(* IEC 61131-3 sources: Codesys/60-let-oktyabrya/src (part 2) *)

(* ---- PRG_AlarmLogSD.st ---- *)
(* ============================================================ *)
(* PRG_AlarmLogSD — ЖУРНАЛЫ НА SD-КАРТУ (3 файла В МЕСЯЦ)        *)
(* ============================================================ *)
(* Пишет на SD три отдельных журнала (чтобы записи не путались): *)
(*   • АВАРИИ     → sAlarmLogPath   (alarms-MM-YYYY.log)         *)
(*   • ИЗМЕНЕНИЯ ПЧ→ sPumpLogPath    (pump_changes-MM-YYYY.log)  *)
(*   • УСТАВКИ    → sSetpointLogPath (setpoints-MM-YYYY.log)     *)
(*                                                              *)
(* === НОВОЕ: ПОМЕСЯЧНЫЕ ФАЙЛЫ ==============================    *)
(* Имя файла содержит месяц и год, поэтому 1-го числа нового     *)
(* месяца путь меняется САМ, и старый автомат (OPEN → если нет   *)
(* файла, то CREATE + BOM) создаёт новый файл без единой строчки *)
(* дополнительной логики. Отдельного «переключателя месяца» нет  *)
(* специально: любая пропущенная граница (ПЛК был выключен,      *)
(* карту вынимали) отрабатывается сама собой при первой записи.  *)
(*                                                              *)
(* === НОВОЕ: КОНТРОЛЬ МЕСТА ================================    *)
(* FB_SdSpaceGuard раз в tSdCheckPeriod (по умолчанию час), при  *)
(* смене месяца и после серии неудачных записей удаляет три файла *)
(* самого старого месяца, если журналы переросли квоту:            *)
(*     квота = ёмкость карты − 100 МБ резерва − чужие файлы        *)
(* Файл текущего месяца удалить нельзя ни при каких условиях.      *)
(*                                                               *)
(* ЁМКОСТЬ КАРТЫ ОПРЕДЕЛЯЕТСЯ АВТОМАТИЧЕСКИ — FB_SdCardSize        *)
(* читает размер раздела у ядра (/sys/block/...). Номинал из       *)
(* выпадающего списка на экране (iSdCardSize) — только запасной    *)
(* вариант, если автоопределение не сработало. Кнопок нет.         *)
(*                                                              *)
(* Строка: "чч:мм дд.мм.гггг - текст" (для аварий) либо готовая  *)
(* строка журнала (для ПЧ/уставок). WSTRING/UTF-16LE + BOM.     *)
(*                                                              *)
(* Аварии детектируются здесь СТРОГО ПО ФРОНТУ FALSE→TRUE: пока  *)
(* авария висит, повторных записей нет. Изменения ПЧ/уставок     *)
(* кладут строку в глобальные очереди GVL_Fountain.awsSdPumpQ /  *)
(* awsSdSetpQ прямо из F_PumpLogWrite / F_FountainLogWrite —      *)
(* здесь мы их только забираем и пишем в файл.                   *)
(*                                                              *)
(* Один конечный автомат обслуживает по очереди все три файла    *)
(* (приоритет: аварии → ПЧ → уставки). ФБ CAA File асинхронные.  *)
(* Пока сторож места занят (fbGuard.xBusy) — новая строка не     *)
(* начинается, строки ждут в очередях.                           *)
(*                                                              *)
(* ТРЕБОВАНИЯ: библиотека CAA File (тип FILE.CAA.HANDLE), карта   *)
(* SD FAT16/FAT32 MBR, путь /mnt/ufs/media/mmcblk0p1/.           *)
(* ============================================================ *)
PROGRAM PRG_AlarmLogSD
VAR CONSTANT
    cAlarmCnt       : INT := 11;   // сколько аварий отслеживаем
    cQSize          : INT := 20;   // глубина очереди строк
    cWriteFailForce : INT := 3;    // столько неудачных записей подряд =
                                   // карта полна → удалить старый месяц
END_VAR
VAR
    (* --- Аварии: состояние + названия --- *)
    axAlarmNow  : ARRAY[1..cAlarmCnt] OF BOOL;
    axAlarmPrev : ARRAY[1..cAlarmCnt] OF BOOL;
    awsAlarmName : ARRAY[1..cAlarmCnt] OF WSTRING(60) := [
        "Сухой ход",
        "Сухой ход реле",
        "Клапан добора реле",
        "Насосы фонтана реле",
        "Подсветка реле",
        "Фильтрация реле (ручной режим)",
        "Связь ПЧ1",
        "Связь ПЧ2",
        "Связь ПЧ3",
        "Связь МВ-Д",
        "Связь МУ"];

    (* --- Локальная очередь аварий (сырые строки, без CRLF) --- *)
    awsAlarmQ : ARRAY[1..cQSize] OF WSTRING(120);
    iAQHead : INT;  iAQTail : INT;  iAQCount : INT;

    (* --- Конечный автомат записи --- *)
    iState     : INT;   // 0=IDLE 1=OPEN 2=CREATE 6=BOM 3=WRITE 4=FLUSH 5=CLOSE 9=DROP
    wsLineOut  : WSTRING(122);
    sActivePath : STRING(80);
    wBom       : WORD := 16#FEFF;   // BOM UTF-16LE (байты FF FE)

    (* --- ФБ CAA File --- *)
    fbFileOpen  : FILE.Open;
    fbFileWrite : FILE.Write;
    fbFileFlush : FILE.Flush;
    fbFileClose : FILE.Close;
    hFile       : FILE.CAA.HANDLE;

    iWrittenCnt : INT;
    iDroppedCnt : INT;

    i          : INT;
    wsTimeStamp : WSTRING(24);
    wsHH : WSTRING(4);  wsMM : WSTRING(4);
    wsDD : WSTRING(4);  wsMo : WSTRING(4);  wsYY : WSTRING(6);

    (* --- Помесячные файлы --- *)
    iLogYear      : INT;    // год/месяц, в которые сейчас пишем
    iLogMonth     : INT;
    iLogYearPrev  : INT;    // 0 при старте → пути соберутся в 1-м же цикле
    iLogMonthPrev : INT;

    (* --- Сторож места на карте --- *)
    fbGuard         : FB_SdSpaceGuard;
    fbCardSize      : FB_SdCardSize;   // автоопределение ёмкости карты
    tonSdCheck      : TON;
    xGuardTrig      : BOOL;
    xGuardStart     : BOOL;
    xCapTrig        : BOOL;   // перечитать ёмкость карты
    xGuardForceAuto : BOOL;   // авто-форс: карта полна (серия отказов записи)
    iWriteFailCnt   : INT;    // неудачных записей подряд
END_VAR

(* ============================================================ *)
(* 1. КАРТА АВАРИЙ (порядок = порядок названий)                 *)
(* ============================================================ *)
axAlarmNow[1]  := xDryRunAlarm;
axAlarmNow[2]  := xDryRunRelayAlarm;
axAlarmNow[3]  := xDamperRelayAlarm;
axAlarmNow[4]  := xPumpRelayAlarm;
axAlarmNow[5]  := xLightRelayAlarm;
axAlarmNow[6]  := xNfManualRelayAlarm;
axAlarmNow[7]  := xPumpCommError[1];
axAlarmNow[8]  := xPumpCommError[2];
axAlarmNow[9]  := xPumpCommError[3];
axAlarmNow[10] := xMV110_Error;
axAlarmNow[11] := xMU110_Error;

(* ============================================================ *)
(* 2. МЕТКА ВРЕМЕНИ "чч:мм дд.мм.гггг"                          *)
(* ============================================================ *)
wsHH := INT_TO_WSTRING(iCurrentHour);   IF iCurrentHour   < 10 THEN wsHH := WCONCAT("0", wsHH); END_IF;
wsMM := INT_TO_WSTRING(iCurrentMinute); IF iCurrentMinute < 10 THEN wsMM := WCONCAT("0", wsMM); END_IF;
wsDD := INT_TO_WSTRING(iCurrentDay);    IF iCurrentDay    < 10 THEN wsDD := WCONCAT("0", wsDD); END_IF;
wsMo := INT_TO_WSTRING(iCurrentMonth);  IF iCurrentMonth  < 10 THEN wsMo := WCONCAT("0", wsMo); END_IF;
wsYY := INT_TO_WSTRING(iCurrentYear);
wsTimeStamp := WCONCAT(wsHH, WCONCAT(":", WCONCAT(wsMM, WCONCAT(" ",
               WCONCAT(wsDD, WCONCAT(".", WCONCAT(wsMo, WCONCAT(".", wsYY))))))));

(* ============================================================ *)
(* 3. ФРОНТ АВАРИИ → строка в локальную очередь аварий          *)
(* ============================================================ *)
FOR i := 1 TO cAlarmCnt DO
    IF axAlarmNow[i] AND NOT axAlarmPrev[i] THEN
        IF xAlarmLogSDEnable THEN
            IF iAQCount < cQSize THEN
                iAQTail := (iAQTail MOD cQSize) + 1;
                awsAlarmQ[iAQTail] := WCONCAT(wsTimeStamp, WCONCAT(" - ", awsAlarmName[i]));
                iAQCount := iAQCount + 1;
            ELSE
                iDroppedCnt := iDroppedCnt + 1;
            END_IF;
        END_IF;
    END_IF;
    axAlarmPrev[i] := axAlarmNow[i];
END_FOR;

(* ============================================================ *)
(* 4. ПУТИ ФАЙЛОВ ТЕКУЩЕГО МЕСЯЦА                               *)
(* ============================================================ *)
(* Если RTC ещё не готов или сбит (села батарейка) — год выйдет  *)
(* за 2000..2199. Писать в "alarms-01-1970.log" нельзя (такой     *)
(* месяц не разберётся обратно и файл станет неудаляемым), поэтому*)
(* весь «бесчасовой» период сваливаем в один файл 01-2000. Он     *)
(* заведомо самый старый по ключу, то есть удалится первым, когда *)
(* место кончится, — и при этом защищён как «текущий», пока RTC   *)
(* не починят.                                                   *)
IF iCurrentYear >= 2000 AND iCurrentYear <= 2199
   AND iCurrentMonth >= 1 AND iCurrentMonth <= 12 THEN
    iLogYear  := iCurrentYear;
    iLogMonth := iCurrentMonth;
    xSdRtcBad := FALSE;
ELSE
    iLogYear  := 2000;
    iLogMonth := 1;
    xSdRtcBad := TRUE;
END_IF;

IF iLogYear <> iLogYearPrev OR iLogMonth <> iLogMonthPrev THEN
    sAlarmLogPath    := F_SdLogPath(sSdLogDir, sAlarmLogPrefix, iLogYear, iLogMonth);
    sPumpLogPath     := F_SdLogPath(sSdLogDir, sPumpLogPrefix,  iLogYear, iLogMonth);
    sSetpointLogPath := F_SdLogPath(sSdLogDir, sSetpLogPrefix,  iLogYear, iLogMonth);
    iLogYearPrev     := iLogYear;
    iLogMonthPrev    := iLogMonth;
    xGuardTrig       := TRUE;    // новый месяц — сразу проверить место
    xCapTrig         := TRUE;    // и заодно перечитать ёмкость карты
END_IF;

(* ============================================================ *)
(* 5. СТОРОЖ МЕСТА НА КАРТЕ                                     *)
(* ============================================================ *)
(* Периодический тик (самосброс: Q взводится на 1 цикл за период) *)
tonSdCheck(IN := NOT tonSdCheck.Q, PT := tSdCheckPeriod);
IF tonSdCheck.Q THEN
    xCapTrig   := TRUE;
    xGuardTrig := TRUE;
END_IF;

(* --- ЁМКОСТЬ КАРТЫ ---                                           *)
(* Сначала пробуем определить её САМИ (FB_SdCardSize читает размер *)
(* раздела у ядра). Получилось — номинал из списка не нужен вообще. *)
(* Не получилось — берём выбранный на экране номинал.               *)
fbCardSize(xTrigger := xCapTrig AND (iState = 0) AND NOT fbGuard.xBusy,
           sSysPath := sSdCardSysPath);
IF fbCardSize.xBusy THEN
    xCapTrig := FALSE;
END_IF;

xSdCapAuto       := fbCardSize.xValid;
udiSdCapAutoMB   := fbCardSize.udiCapacityMB;
udiSdCardSectors := fbCardSize.udiSectors;

IF iSdCardSize < 0 THEN iSdCardSize := 0; END_IF;
IF iSdCardSize > 6 THEN iSdCardSize := 6; END_IF;

IF xSdCapAuto THEN
    udiSdUsableMB := udiSdCapAutoMB;
ELSE
    udiSdUsableMB := audiSdCardMB[iSdCardSize];
END_IF;

(* АВАРИЙНЫЙ ФОРС. Если запись не проходит подряд cWriteFailForce  *)
(* раз — карта реально полна, что бы ни говорил расчёт по номиналу *)
(* (например, в списке выбрали 32 ГБ, а стоит карта на 16). Тогда  *)
(* удаляем самый старый месяц безусловно. Одиночный сбой записи к  *)
(* удалению НЕ приводит — только серия подряд.                     *)
IF iWriteFailCnt >= cWriteFailForce THEN
    xGuardTrig      := TRUE;
    xGuardForceAuto := TRUE;
    iWriteFailCnt   := 0;
END_IF;

(* Запускаем сторожа ТОЛЬКО когда автомат записи стоит в IDLE:     *)
(* так исключено удаление файла при открытом дескрипторе.          *)
xGuardStart := xGuardTrig AND xAlarmLogSDEnable
               AND (iState = 0) AND NOT fbGuard.xBusy AND NOT fbCardSize.xBusy;

fbGuard(xTrigger      := xGuardStart,
        xForce        := xGuardForceAuto,
        sDir          := sSdLogDir,
        sPrefix1      := sAlarmLogPrefix,
        sPrefix2      := sPumpLogPrefix,
        sPrefix3      := sSetpLogPrefix,
        udiUsableMB   := udiSdUsableMB,
        udiFreeMinMB  := udiSdFreeMinMB,
        iCurYear      := iLogYear,
        iCurMonth     := iLogMonth);

IF fbGuard.xBusy THEN
    xGuardTrig      := FALSE;
    xGuardForceAuto := FALSE;
END_IF;

(* Диагностика на экран *)
udiSdQuotaMB       := fbGuard.udiQuotaMB;
udiSdOursMB        := fbGuard.udiOursMB;
udiSdUsedMB        := fbGuard.udiUsedMB;
udiSdForeignMB     := fbGuard.udiForeignMB;
udiSdOldestMB      := fbGuard.udiOldestMB;
xSdNothingToDelete := fbGuard.xNothingToDelete;
xSdLogQuotaStop    := fbGuard.xQuotaStop;
xSdCleanupFault    := fbGuard.xFault;
iSdDeletedTotal    := fbGuard.iDeletedTotal;
sSdLastDeleted     := fbGuard.sLastDeleted;

(* ============================================================ *)
(* 6. КОНЕЧНЫЙ АВТОМАТ: пишет по очереди 3 файла                *)
(*    приоритет: аварии → изменения ПЧ → уставки               *)
(* ============================================================ *)
(* Запись стоит, пока сторож занят (иначе он удалял бы файл с    *)
(* открытым дескриптором) ИЛИ пока поднят xQuotaStop — последний *)
(* рубеж защиты карты: наши журналы упёрлись в квоту, а удалять   *)
(* уже нечего. Строки при этом копятся в очередях, лишние         *)
(* считаются в iDroppedCnt; журналы на экране ведутся как обычно. *)
IF NOT fbGuard.xBusy AND NOT fbCardSize.xBusy AND NOT fbGuard.xQuotaStop THEN

CASE iState OF

    0:  (* IDLE — выбрать непустую очередь, взять строку, начать *)
        IF xAlarmLogSDEnable THEN
            IF iAQCount > 0 THEN
                iAQHead := (iAQHead MOD cQSize) + 1;
                wsLineOut := WCONCAT(awsAlarmQ[iAQHead], "$R$N");
                iAQCount := iAQCount - 1;
                sActivePath := sAlarmLogPath;
                iState := 1;
            ELSIF iSdPumpQCount > 0 THEN
                iSdPumpQHead := (iSdPumpQHead MOD 20) + 1;
                wsLineOut := WCONCAT(awsSdPumpQ[iSdPumpQHead], "$R$N");
                iSdPumpQCount := iSdPumpQCount - 1;
                sActivePath := sPumpLogPath;
                iState := 1;
            ELSIF iSdSetpQCount > 0 THEN
                iSdSetpQHead := (iSdSetpQHead MOD 20) + 1;
                wsLineOut := WCONCAT(awsSdSetpQ[iSdSetpQHead], "$R$N");
                iSdSetpQCount := iSdSetpQCount - 1;
                sActivePath := sSetpointLogPath;
                iState := 1;
            END_IF;
        END_IF;

    1:  (* OPEN на дозапись *)
        fbFileOpen(xExecute := TRUE, sFileName := sActivePath, eFileMode := FILE.MODE.MAPPD);
        IF fbFileOpen.xDone THEN
            hFile := fbFileOpen.hFile;
            fbFileOpen(xExecute := FALSE);
            iState := 3;
        ELSIF fbFileOpen.xError THEN
            IF fbFileOpen.eError = FILE.ERROR.NOT_EXIST THEN
                fbFileOpen(xExecute := FALSE);
                iState := 2;
            ELSE
                fbFileOpen(xExecute := FALSE);
                iState := 9;
            END_IF;
        END_IF;

    2:  (* CREATE — MWRITE создаёт файл *)
        fbFileOpen(xExecute := TRUE, sFileName := sActivePath, eFileMode := FILE.MODE.MWRITE);
        IF fbFileOpen.xDone THEN
            hFile := fbFileOpen.hFile;
            fbFileOpen(xExecute := FALSE);
            iState := 6;
        ELSIF fbFileOpen.xError THEN
            fbFileOpen(xExecute := FALSE);
            iState := 9;
        END_IF;

    6:  (* WRITE_BOM — метка UTF-16LE в начало нового файла *)
        fbFileWrite(xExecute := TRUE, hFile := hFile, pBuffer := ADR(wBom), szSize := UDINT#2);
        IF fbFileWrite.xDone THEN
            fbFileWrite(xExecute := FALSE);
            iState := 3;
        ELSIF fbFileWrite.xError THEN
            fbFileWrite(xExecute := FALSE);
            xSdWriteFault := TRUE;
            xGuardTrig    := TRUE;
            iWriteFailCnt := iWriteFailCnt + 1;      // не пишется — проверить место
            iState := 5;
        END_IF;

    3:  (* WRITE — строка WSTRING, размер = WLEN*2 байт *)
        fbFileWrite(xExecute := TRUE, hFile := hFile,
                    pBuffer := ADR(wsLineOut), szSize := INT_TO_UDINT(WLEN(wsLineOut) * 2));
        IF fbFileWrite.xDone THEN
            fbFileWrite(xExecute := FALSE);
            iWrittenCnt := iWrittenCnt + 1;
            xSdWriteFault := FALSE;
            iWriteFailCnt := 0;         // запись прошла — серия отказов сброшена
            iState := 4;
        ELSIF fbFileWrite.xError THEN
            fbFileWrite(xExecute := FALSE);
            xSdWriteFault := TRUE;
            xGuardTrig    := TRUE;
            iWriteFailCnt := iWriteFailCnt + 1;
            iState := 5;
        END_IF;

    4:  (* FLUSH *)
        fbFileFlush(xExecute := TRUE, hFile := hFile);
        IF fbFileFlush.xDone OR fbFileFlush.xError THEN
            fbFileFlush(xExecute := FALSE);
            iState := 5;
        END_IF;

    5:  (* CLOSE *)
        fbFileClose(xExecute := TRUE, hFile := hFile);
        IF fbFileClose.xDone OR fbFileClose.xError THEN
            fbFileClose(xExecute := FALSE);
            iState := 0;
        END_IF;

    9:  (* DROP — ошибка открытия/создания, едем дальше *)
        xSdWriteFault := TRUE;
        xGuardTrig    := TRUE;
        iWriteFailCnt := iWriteFailCnt + 1;
        iState := 0;

END_CASE;

END_IF;

(* ---- PRG_Errors.st ---- *)
(* ============================================================ *)
(* PRG_Errors — ЕДИНЫЙ подсчёт аварий + статус системы          *)
(* Проект "60 Лет Октября" (на основе ДДЮТ / Саки Пруд).         *)
(* ============================================================ *)
PROGRAM PRG_Errors
VAR
    i : INT;
END_VAR

iErrors         := 0;
iErrorsPumps    := 0;
iErrorsModules  := 0;
iErrorsFountain := 0;
iWorkCount      := 0;
iStopCount      := 0;

(* ============================================================ *)
(* 1. АВАРИИ НАСОСОВ ПЧ (счётчик iErrorsPumps)                  *)
(* ============================================================ *)
FOR i := 1 TO cPumpCount DO
    IF xPumpAlarm[i] AND NOT xPumpCommError[i] THEN
        iErrorsPumps := iErrorsPumps + 1;
    END_IF;
    IF xPumpWork[i] THEN iWorkCount := iWorkCount + 1; END_IF;
    IF xPumpStop[i] THEN iStopCount := iStopCount + 1; END_IF;
END_FOR;

(* ============================================================ *)
(* 2. АВАРИИ СВЯЗИ МОДУЛЕЙ (счётчик iErrorsModules)              *)
(* ============================================================ *)
FOR i := 1 TO cPumpCount DO
    IF xPumpCommError[i] THEN
        iErrorsModules := iErrorsModules + 1;
    END_IF;
END_FOR;
IF xMV110_Error THEN iErrorsModules := iErrorsModules + 1; END_IF;
IF xMU110_Error THEN iErrorsModules := iErrorsModules + 1; END_IF;

(* ============================================================ *)
(* 3. АВАРИИ АВТОМАТИКИ ФОНТАНА (iErrorsFountain)                *)
(* ⚠️ Сухой ход учитывается первым по смыслу (см. sAlarmCauses      *)
(* в PRG_Fountain.st, блок 11, где он тоже первый в строке).        *)
(* Опасная ситуация (сухой ход + ручная фильтрация) сюда НЕ         *)
(* включается — это не блокирующая авария, а рекомендация            *)
(* оператору, у неё своя отдельная лампа/диалог (xShowDangerDialog). *)
(* ============================================================ *)
IF xDryRunAlarm        THEN iErrorsFountain := iErrorsFountain + 1; END_IF;  // сухой ход — САМАЯ ОПАСНАЯ
IF xDryRunRelayAlarm   THEN iErrorsFountain := iErrorsFountain + 1; END_IF;  // реле сухого хода (DO1/DI8)
IF xDamperRelayAlarm   THEN iErrorsFountain := iErrorsFountain + 1; END_IF;  // реле клапана добора (DO4/DI6)
IF xPumpRelayAlarm     THEN iErrorsFountain := iErrorsFountain + 1; END_IF;  // реле насосов фонтана (DO2/DI9)
IF xLightRelayAlarm    THEN iErrorsFountain := iErrorsFountain + 1; END_IF;  // реле подсветки (DO3/DI10)
IF xNfManualRelayAlarm THEN iErrorsFountain := iErrorsFountain + 1; END_IF;  // реле фильтрации, ручной режим

(* ============================================================ *)
(* 4. ОБЩИЙ СЧЁТЧИК ВСЕХ АВАРИЙ + ЕДИНЫЙ ФЛАГ                    *)
(* ============================================================ *)
iErrors   := iErrorsPumps + iErrorsModules + iErrorsFountain;
xAnyAlarm := (iErrors > 0);

xSystemState := NOT xAnyAlarm;
IF xSystemState THEN
    sSystemStateText := "Система: ОК";
ELSE
    sSystemStateText := "Авария";
END_IF;

(* ---- PRG_Fountain.st ---- *)
PROGRAM PRG_Fountain
(* ============================================================ *)
(* PRG_Fountain — автоматика "60 Лет Октября"                   *)
(* (на основе ДДЮТ / Саки Пруд)                                 *)
(* ============================================================ *)
VAR
    dwUtcTime : DWORD;
    sysTime   : SYSTIMEDATE;
    rtcResult : DWORD;

    fbTimeZone : FB_TimeZoneSelect;
    fbSunset : FB_SunsetRelay;
    fbSchedule : FB_FountainSchedule;

    tonBlinkFastOff : TON;
    tonBlinkSlowOff : TON;

    tonNfContinuous : TON;

    (* 60ЛО: таймеры проверки реле (обрыв/залипание) *)
    tonDryRunRelayAlarm : TON;   // DO1 vs DI8, 2с
    tonDamperRelayAlarm : TON;   // DO4 vs DI6, 20с (процесс не мгновенный)
    tonPumpRelayAlarm   : TON;   // DO2 vs DI9, 2с
    tonLightRelayAlarm  : TON;   // DO3 vs DI10, 2с
    tonNfManualRelayAlarm : TON; // ручной режим (DI12) и DI7=0, 2с

    iClearIdx : INT;

    tonFountainLogClearedMsg : TON;
    tonFountainLogPassBadMsg : TON;
    tonPumpLogClearedMsg     : TON;
    tonPumpLogPassBadMsg     : TON;
END_VAR

(* ============================================================ *)
(* 1. ЧТЕНИЕ СИСТЕМНОГО ВРЕМЕНИ (RTC) — БЕЗ ИЗМЕНЕНИЙ            *)
(* ============================================================ *)
dwUtcTime := SysTimeRtcGet(pResult := rtcResult);
dwUtcTime := dwUtcTime + INT_TO_DWORD(iTimeZoneOffsetSec);
rtcResult := SysTimeRtcConvertUtcToDate(dwTimestampUtc := dwUtcTime, pDate := sysTime);
iCurrentYear         := WORD_TO_INT(sysTime.wYear);
iCurrentMonth        := WORD_TO_INT(sysTime.wMonth);
iCurrentDay          := WORD_TO_INT(sysTime.wDay);
iCurrentHour         := WORD_TO_INT(sysTime.wHour);
iCurrentMinute       := WORD_TO_INT(sysTime.wMinute);
iCurrentSecond       := WORD_TO_INT(sysTime.wSecond);
iCurrentTotalMinutes := iCurrentHour * 60 + iCurrentMinute;

IF iCurrentDay < 10 THEN
    sCurrentDateStr := WCONCAT("0", INT_TO_WSTRING(iCurrentDay));
ELSE
    sCurrentDateStr := INT_TO_WSTRING(iCurrentDay);
END_IF;
IF iCurrentMonth < 10 THEN
    sCurrentDateStr := WCONCAT(sCurrentDateStr, WCONCAT(".0", INT_TO_WSTRING(iCurrentMonth)));
ELSE
    sCurrentDateStr := WCONCAT(sCurrentDateStr, WCONCAT(".", INT_TO_WSTRING(iCurrentMonth)));
END_IF;
sCurrentDateStr := WCONCAT(sCurrentDateStr, WCONCAT(".", INT_TO_WSTRING(iCurrentYear)));

(* ============================================================ *)
(* 2. РАСПАКОВКА ВХОДОВ DI — 60ЛО: НОВАЯ КАРТА                    *)
(* ============================================================ *)
xPump1Work := xDI[1];    // ПЧ1 (информационный)
xPump2Work := xDI[2];    // ПЧ2 (информационный)
xPump3Work := xDI[3];    // ПЧ3 (информационный, НОВЫЙ)
xDryRunOk       := xDI[4];    // сухой ход от Мусидоры, 1=норма
xDamperCmdRaw   := xDI[5];    // пуск добора от Мусидоры
xDamperRelayFb  := xDI[6];    // подтверждение положения клапана добора
xNfWork         := xDI[7];    // контактор фильтрации
xDryRunRelayFb  := xDI[8];    // подтверждение реле сухого хода
xPumpRelayFb    := xDI[9];    // подтверждение работы насосов фонтана
xLightRelayFb   := xDI[10];   // подтверждение работы подсветки
xNfAutoSwitch   := xDI[11];   // ручка режима фильтрации = АВТО
xNfManualSwitch := xDI[12];   // ручка режима фильтрации = РУЧНОЙ

(* ============================================================ *)
(* 2а. РЕЖИМЫ — СЕЛЕКТОР ДЛЯ СВЕТА И НАСОСОВ ФОНТАНА             *)
(* ============================================================ *)
(*   0 = Ручной пуск (принудительно вкл, минуя автоматику)         *)
(*   1 = Выкл (запрет)                                             *)
(*   2 = Авто (штатная логика по расписанию)                       *)

(* Насосы фонтана *)
IF iPumpSelect = 0 THEN
    xManualPermissionNasos := FALSE;
    xPumpsForceOn          := TRUE;
ELSIF iPumpSelect = 2 THEN
    xManualPermissionNasos := TRUE;
    xPumpsForceOn          := FALSE;
ELSE
    xManualPermissionNasos := FALSE;
    xPumpsForceOn          := FALSE;
END_IF;

xPumpOuterForcedOn  := (iPumpSelect = 0);
xPumpOuterForcedOff := (iPumpSelect = 1);

(* Свет *)
IF iLightSelect = 0 THEN
    xLightEnable  := FALSE;
    xLightForceOn := TRUE;
ELSIF iLightSelect = 2 THEN
    xLightEnable  := TRUE;
    xLightForceOn := FALSE;
ELSE
    xLightEnable  := FALSE;
    xLightForceOn := FALSE;
END_IF;

xLightOuterForcedOn  := (iLightSelect = 0);
xLightOuterForcedOff := (iLightSelect = 1);

(* ============================================================ *)
(* 3. СУХОЙ ХОД + ПРОВЕРКА РЕЛЕ (2с)                             *)
(* ============================================================ *)
xDryRunAlarm := NOT xDryRunOk;    // ЖИВАЯ, НЕ защёлка. САМАЯ ПЕРВАЯ авария в списке!

(* === 60ЛО:ИСПРАВЛЕНО (баг) === Раньше здесь сравнивался xDO[1]  *)
(* — но он ещё не переписан на этом цикле (запись в блоке 15,     *)
(* позже), т.е. сравнение шло со значением ПРОШЛОГО цикла.        *)
(* xDryRunOk — то же самое значение, которое уйдёт на DO1 в этом   *)
(* же цикле (просто зеркало DI4→DO1), поэтому сравниваем с ним     *)
(* напрямую — без задержки на цикл.                                *)
tonDryRunRelayAlarm(IN := xDryRunOk <> xDryRunRelayFb, PT := T#2S);
IF tonDryRunRelayAlarm.Q THEN
    xDryRunRelayAlarm := TRUE;
END_IF;
IF xAlarmReset THEN
    xDryRunRelayAlarm := FALSE;
    tonDryRunRelayAlarm(IN := FALSE, PT := T#2S);
END_IF;

(* ============================================================ *)
(* 4. КЛАПАН ДОБОРА — ЗЕРКАЛО DI5→DO4, проверка реле 20с          *)
(* ============================================================ *)
IF xDamperRelayFb THEN
    sDamperPosition := "Открыт";
ELSE
    sDamperPosition := "Закрыт";
END_IF;

tonDamperRelayAlarm(IN := xDamperCmdRaw <> xDamperRelayFb, PT := T#20S);
IF tonDamperRelayAlarm.Q THEN
    xDamperRelayAlarm := TRUE;
END_IF;
IF xAlarmReset THEN
    xDamperRelayAlarm := FALSE;
    tonDamperRelayAlarm(IN := FALSE, PT := T#20S);
END_IF;

(* ============================================================ *)
(* 5. ФИЛЬТРАЦИЯ — режим/авария реле (2с)                        *)
(* ============================================================ *)
tonNfManualRelayAlarm(IN := xNfManualSwitch AND NOT xNfWork, PT := T#2S);
IF tonNfManualRelayAlarm.Q THEN
    xNfManualRelayAlarm := TRUE;
END_IF;
IF xAlarmReset THEN
    xNfManualRelayAlarm := FALSE;
    tonNfManualRelayAlarm(IN := FALSE, PT := T#2S);
END_IF;

(* === 60ЛО:ИСПРАВЛЕНО (баг компиляции) === Раньше здесь стоял      *)
(* CASE TRUE OF — в CODESYS так писать НЕЛЬЗЯ (метка CASE требует   *)
(* целочисленный литерал, не BOOL). Заменено на обычный IF/ELSIF.   *)
(* Логика: если ни DI11, ни DI12 не активны одновременно — это      *)
(* либо промежуточное положение ручки (если оно физически возможно),*)
(* либо обрыв провода на оба входа — статус "?" сигнализирует       *)
(* оператору о нештатной ситуации, чтобы не осталось старое          *)
(* значение "Авто"/"Ручной" на экране.                               *)
IF xNfAutoSwitch THEN
    sNfModeStatus := "Авто";
ELSIF xNfManualSwitch THEN
    sNfModeStatus := "Ручной";
ELSE
    sNfModeStatus := "?";   // ни один вход не активен — обрыв линии или промежуточное положение
END_IF;

IF xNfWork THEN sNfStatus := "Работает"; ELSE sNfStatus := "Стоп"; END_IF;

(* ============================================================ *)
(* 5а. СЧЁТЧИК ПРОМЫВОК НФ — БЕЗ ИЗМЕНЕНИЙ АЛГОРИТМА             *)
(* ============================================================ *)
IF NOT xNfFirstScanDone THEN
    xNfFirstScanDone := TRUE;
    xNfWorkPrev := xNfWork;
END_IF;

IF xNfHealthy THEN
    iNfFlushStage := 0;
    xNfFlushReady := TRUE;
END_IF;

IF xNfWork AND NOT xNfWorkPrev THEN
    iNfLastOnHour  := iCurrentHour;
    iNfLastOnMin   := iCurrentMinute;
    iNfLastOnDay   := iCurrentDay;
    iNfLastOnMonth := iCurrentMonth;
    iNfLastOnYear  := iCurrentYear;
END_IF;

IF (NOT xNfWork) AND xNfWorkPrev THEN
    iNfJustEndedSec := DINT_TO_INT(TIME_TO_DINT(tonNfContinuous.ET) / 1000);

    IF xNfFlushReady THEN
        IF (iNfJustEndedSec > 60) AND (iNfJustEndedSec < (iFilterMinRunMin * 60)) THEN
            IF iNfFlushStage = 0 THEN
                iNfFlushStage := 1;
            ELSE
                iNfFlushCount  := iNfFlushCount + 1;
                iNfFlushHour   := iCurrentHour;
                iNfFlushMin    := iCurrentMinute;
                iNfFlushDay    := iCurrentDay;
                iNfFlushMonth  := iCurrentMonth;
                iNfFlushYear   := iCurrentYear;
                iNfFlushStage  := 0;
                xNfFlushReady  := FALSE;
            END_IF;
        END_IF;
    END_IF;
END_IF;

xNfWorkPrev := xNfWork;

(* Сброс счётчика промывок — СВОЙ отдельный диалог, НЕ через xAlarmReset. *)
IF xConfirmResetNfFlush THEN
    iNfFlushCount  := 0;
    iNfFlushStage  := 0;
    xNfFlushReady  := TRUE;
    iNfFlushHour   := 0;
    iNfFlushMin    := 0;
    iNfFlushDay    := 0;
    iNfFlushMonth  := 0;
    iNfFlushYear   := 0;
    xAskResetNfFlush     := FALSE;
    xConfirmResetNfFlush := FALSE;
    F_FountainLogWrite("Сброс счётчика промывок НФ");
END_IF;
(* Кнопки на экране: "Сбросить" → xAskResetNfFlush:=TRUE (показать окно);  *)
(* "Подтвердить" → xConfirmResetNfFlush:=TRUE; "Отмена" → xAskResetNfFlush:=FALSE. *)

(* ============================================================ *)
(* 5б. ИСПРАВНОСТЬ НФ — непрерывная наработка, БЕЗ ИЗМЕНЕНИЙ      *)
(* ============================================================ *)
tonNfContinuous(IN := xNfWork,
    PT := DINT_TO_TIME(INT_TO_DINT(iFilterMinRunMin) * 60000));
xNfHealthy := tonNfContinuous.Q;

iNfContinuousRunHour := DINT_TO_INT(TIME_TO_DINT(tonNfContinuous.ET) / 3600000);
iNfContinuousRunMin  := DINT_TO_INT((TIME_TO_DINT(tonNfContinuous.ET) MOD 3600000) / 60000);
iNfContinuousRunSec  := DINT_TO_INT((TIME_TO_DINT(tonNfContinuous.ET) MOD 60000) / 1000);

(* ============================================================ *)
(* 6. РАСЧЁТ ЗАКАТА — NOAA v2, БЕЗ ИЗМЕНЕНИЙ                     *)
(* ============================================================ *)
IF (rSunLongitude > rSunLongitudePrev + 0.01) OR (rSunLongitude < rSunLongitudePrev - 0.01) THEN
    rSunLongitudePrev := rSunLongitude;
    iChoseTimeZone := REAL_TO_INT(rSunLongitude / 15.0) + 11;
    IF iChoseTimeZone > 23 THEN
        iChoseTimeZone := 23;
    ELSIF iChoseTimeZone < 0 THEN
        iChoseTimeZone := 0;
    END_IF;
END_IF;

fbTimeZone(ChoseTimeZone := INT_TO_UDINT(iChoseTimeZone));
rSunTimeZone := fbTimeZone.TimeZone;

IF iSunsetCorrectSigned < 0 THEN
    xSunsetCorrectEarlier := TRUE;
    iSunsetCorrectMin     := -iSunsetCorrectSigned;
ELSE
    xSunsetCorrectEarlier := FALSE;
    iSunsetCorrectMin     := iSunsetCorrectSigned;
END_IF;

fbSunset(
    Latitude           := rSunLatitude,
    Longitude          := rSunLongitude,
    TimeZone           := rSunTimeZone,
    Sunset_Correct     := INT_TO_UDINT(iSunsetCorrectMin),
    Sunset_Earlier     := xSunsetCorrectEarlier,
    Off_Hour_Weekday   := INT_TO_UDINT(iOffHourWeekday),
    Off_Minute_Weekday := INT_TO_UDINT(iOffMinuteWeekday),
    Off_Hour_Weekend   := INT_TO_UDINT(iOffHourWeekend),
    Off_Minute_Weekend := INT_TO_UDINT(iOffMinuteWeekend),
    Sys_Year           := INT_TO_UDINT(iCurrentYear),
    Sys_Month          := INT_TO_UDINT(iCurrentMonth),
    Sys_Day            := INT_TO_UDINT(iCurrentDay),
    Sys_Hour           := INT_TO_UDINT(iCurrentHour),
    Sys_Minute         := INT_TO_UDINT(iCurrentMinute),
    Sys_Sec            := INT_TO_UDINT(iCurrentSecond)
);
xSunsetActive     := fbSunset.Sunset_Auto;
xSunsetCoordError := fbSunset.Err_Coord;
iSunsetHourCalc   := UDINT_TO_INT(fbSunset.Sunset_Hour);
iSunsetMinuteCalc := UDINT_TO_INT(fbSunset.Sunset_Minute);
iSunsetTimeLeftH  := UDINT_TO_INT(fbSunset.Time_Left_H);
iSunsetTimeLeftM  := UDINT_TO_INT(fbSunset.Time_Left_M);
iSunsetDayOfYear  := UDINT_TO_INT(fbSunset.DayOfYear);
xIsWeekend        := fbSunset.IsWeekend;

(* ============================================================ *)
(* 7. РАСПИСАНИЕ СВЕТА/НАСОСОВ — FB_FountainSchedule, БЕЗ ИЗМЕНЕНИЙ *)
(* ============================================================ *)
fbSchedule(
    Sunset_Auto             := fbSunset.Sunset_Auto,
    Sunset_Hour             := fbSunset.Sunset_Hour,
    Sunset_Minute           := fbSunset.Sunset_Minute,
    IsWeekend               := fbSunset.IsWeekend,
    Light_Mode              := INT_TO_UDINT(iLightScheduleMode),
    Light_On_Hour_Weekday   := INT_TO_UDINT(iLightOnHourWeekday),
    Light_On_Minute_Weekday := INT_TO_UDINT(iLightOnMinuteWeekday),
    Light_On_Hour_Weekend   := INT_TO_UDINT(iLightOnHourWeekend),
    Light_On_Minute_Weekend := INT_TO_UDINT(iLightOnMinuteWeekend),
    Off_Hour_Weekday        := INT_TO_UDINT(iOffHourWeekday),
    Off_Minute_Weekday      := INT_TO_UDINT(iOffMinuteWeekday),
    Off_Hour_Weekend        := INT_TO_UDINT(iOffHourWeekend),
    Off_Minute_Weekend      := INT_TO_UDINT(iOffMinuteWeekend),
    Pump_Mode                := INT_TO_UDINT(iPumpScheduleMode),
    Pump_On_Hour_Weekday    := INT_TO_UDINT(iPumpOnHourWeekday),
    Pump_On_Minute_Weekday  := INT_TO_UDINT(iPumpOnMinuteWeekday),
    Pump_On_Hour_Weekend    := INT_TO_UDINT(iPumpOnHourWeekend),
    Pump_On_Minute_Weekend  := INT_TO_UDINT(iPumpOnMinuteWeekend),
    Sys_Hour                := INT_TO_UDINT(iCurrentHour),
    Sys_Minute              := INT_TO_UDINT(iCurrentMinute)
);
xScheduleLightOut      := fbSchedule.Light_Out;
xSchedulePumpOut       := fbSchedule.Pump_Out;
iScheduleLightOnHour   := UDINT_TO_INT(fbSchedule.Light_On_Result_Hour);
iScheduleLightOnMinute := UDINT_TO_INT(fbSchedule.Light_On_Result_Minute);
iScheduleOffHour       := UDINT_TO_INT(fbSchedule.Off_Result_Hour);
iScheduleOffMinute     := UDINT_TO_INT(fbSchedule.Off_Result_Minute);
iSchedulePumpOnHour    := UDINT_TO_INT(fbSchedule.Pump_On_Result_Hour);
iSchedulePumpOnMinute  := UDINT_TO_INT(fbSchedule.Pump_On_Result_Minute);

xLightShowInputFields   := fbSchedule.Light_ShowInputFields;
xLightShowComputedTime  := fbSchedule.Light_ShowComputedTime;
xLightShowAlwaysOnText  := fbSchedule.Light_ShowAlwaysOnText;
xLightShowAlwaysOffText := fbSchedule.Light_ShowAlwaysOffText;
xPumpShowInputFields    := fbSchedule.Pump_ShowInputFields;
xPumpShowComputedTime   := fbSchedule.Pump_ShowComputedTime;
xPumpShowAlwaysOnText   := fbSchedule.Pump_ShowAlwaysOnText;
xPumpShowAlwaysOffText  := fbSchedule.Pump_ShowAlwaysOffText;
xOffTimeVisible         := fbSchedule.Off_Time_Visible;

(* ============================================================ *)
(* 8. ГЕНЕРАТОРЫ МИГАНИЯ — БЕЗ ИЗМЕНЕНИЙ                          *)
(* ============================================================ *)
tonBlinkFastOff(IN := xBlinkFast, PT := T#20MS);
IF tonBlinkFastOff.Q THEN xBlinkFast := FALSE; END_IF;
IF NOT xBlinkFast AND NOT tonBlinkFastOff.IN THEN xBlinkFast := TRUE; END_IF;

tonBlinkSlowOff(IN := xBlinkSlow, PT := T#100MS);
IF tonBlinkSlowOff.Q THEN xBlinkSlow := FALSE; END_IF;
IF NOT xBlinkSlow AND NOT tonBlinkSlowOff.IN THEN xBlinkSlow := TRUE; END_IF;

(* ============================================================ *)
(* 9. НАСОСЫ ФОНТАНА (DO2) + проверка реле (2с)                  *)
(* ============================================================ *)
xPumpsCmd := xVseSist AND NOT xDryRunAlarm AND xManualPermissionNasos AND xSchedulePumpOut;
IF xPumpsForceOn THEN
    xPumpsCmd := TRUE;   // ручной пуск — минуя все запреты
END_IF;

tonPumpRelayAlarm(IN := xPumpsCmd <> xPumpRelayFb, PT := T#2S);
IF tonPumpRelayAlarm.Q THEN
    xPumpRelayAlarm := TRUE;
END_IF;
IF xAlarmReset THEN
    xPumpRelayAlarm := FALSE;
    tonPumpRelayAlarm(IN := FALSE, PT := T#2S);
END_IF;

CASE iPumpSelect OF
    0: sPermissionStatus := "Ручной пуск";
    2: sPermissionStatus := "Авто";
ELSE
    sPermissionStatus := "Выкл";
END_CASE;

(* ============================================================ *)
(* 10. ПОДСВЕТКА (DO3) + проверка реле (2с)                      *)
(* ============================================================ *)
xLightCmd := NOT xDryRunAlarm AND xVseSist AND xLightEnable AND xScheduleLightOut;
IF xLightForceOn THEN
    xLightCmd := TRUE;
END_IF;

tonLightRelayAlarm(IN := xLightCmd <> xLightRelayFb, PT := T#2S);
IF tonLightRelayAlarm.Q THEN
    xLightRelayAlarm := TRUE;
END_IF;
IF xAlarmReset THEN
    xLightRelayAlarm := FALSE;
    tonLightRelayAlarm(IN := FALSE, PT := T#2S);
END_IF;

CASE iLightSelect OF
    0: sLightStatus := "Ручной пуск";
    2: sLightStatus := "Авто (закат)";
ELSE
    sLightStatus := "Выкл";
END_CASE;

(* ============================================================ *)
(* 11. ОБЩАЯ АВАРИЯ + СТРОКА ПРИЧИН — сухой ход ПЕРВЫМ            *)
(* ============================================================ *)
(* === 60ЛО:ИЗМЕНЕНО === "Опасная ситуация" (сухой ход + ручная  *)
(* фильтрация) СЮДА больше не выводится — у неё СВОЯ отдельная    *)
(* лампа/диалог (xShowDangerDialog, блок 12). Если добавить её     *)
(* и в общий список причин, счётчик iErrors (PRG_Errors.st) и      *)
(* текст sAlarmCauses разойдутся, т.к. в счётчик она не входит      *)
(* (не блокирующая авария, а рекомендация оператору).               *)
xAlarmFountain := xDryRunAlarm
              OR xDryRunRelayAlarm
              OR xDamperRelayAlarm
              OR xPumpRelayAlarm
              OR xLightRelayAlarm
              OR xNfManualRelayAlarm;

sAlarmCauses := "";
IF xDryRunAlarm         THEN sAlarmCauses := WCONCAT(sAlarmCauses, "Сухой ход, ");            END_IF;
IF xDryRunRelayAlarm    THEN sAlarmCauses := WCONCAT(sAlarmCauses, "Сухой ход реле, ");        END_IF;
IF xDamperRelayAlarm    THEN sAlarmCauses := WCONCAT(sAlarmCauses, "Клапан добора реле, ");    END_IF;
IF xPumpRelayAlarm      THEN sAlarmCauses := WCONCAT(sAlarmCauses, "Насосы фонтана реле, ");   END_IF;
IF xLightRelayAlarm     THEN sAlarmCauses := WCONCAT(sAlarmCauses, "Подсветка реле, ");        END_IF;
IF xNfManualRelayAlarm  THEN sAlarmCauses := WCONCAT(sAlarmCauses, "Фильтрация реле (ручной режим), "); END_IF;
IF xPumpCommError[1]    THEN sAlarmCauses := WCONCAT(sAlarmCauses, "Связь ПЧ1, ");             END_IF;
IF xPumpCommError[2]    THEN sAlarmCauses := WCONCAT(sAlarmCauses, "Связь ПЧ2, ");             END_IF;
IF xPumpCommError[3]    THEN sAlarmCauses := WCONCAT(sAlarmCauses, "Связь ПЧ3, ");             END_IF;
IF xMV110_Error         THEN sAlarmCauses := WCONCAT(sAlarmCauses, "Связь МВ-Д, ");            END_IF;
IF xMU110_Error         THEN sAlarmCauses := WCONCAT(sAlarmCauses, "Связь МУ, ");              END_IF;
IF sAlarmCauses = ""    THEN sAlarmCauses := "Нет аварий";                                    END_IF;

IF xAlarmReset THEN
    xAlarmReset := FALSE;
END_IF;

IF xAlarmFountain THEN sAlarmStopStatus := "Да"; ELSE sAlarmStopStatus := "Нет"; END_IF;

(* ============================================================ *)
(* 12. ОПАСНАЯ СИТУАЦИЯ: СУХОЙ ХОД + РУЧНАЯ ФИЛЬТРАЦИЯ            *)
(* ============================================================ *)
(* Ничего не блокируем — только напоминание. Показ по фронту       *)
(* появления, кнопка "ОК" на диалоге выполняет ОДНУ строку:         *)
(*   GVL_Fountain.xConfirmDangerDialog := TRUE;                     *)
(* Если ситуация уйдёт и появится заново — диалог покажется снова.  *)
xDangerCondition := xDryRunAlarm AND xNfManualSwitch;

IF xDangerCondition AND NOT xDangerCondition_Prev THEN
    xShowDangerDialog := TRUE;
END_IF;
IF xConfirmDangerDialog THEN
    xShowDangerDialog    := FALSE;
    xConfirmDangerDialog := FALSE;
END_IF;
xDangerCondition_Prev := xDangerCondition;

(* ============================================================ *)
(* 13. ЖУРНАЛ ИЗМЕНЕНИЙ ПАРАМЕТРОВ ФОНТАНА — СПИСОК СОКРАЩЁН      *)
(* ============================================================ *)
IF xFountainLogPinSubmit THEN
    xFountainLogPinSubmit := FALSE;
    IF iFountainLogPinEntry = iAdminPassCorrect THEN
        xFountainLogClear      := TRUE;
        xAskClearFountainLog   := FALSE;
        xFountainLogClearedMsg := TRUE;
    ELSE
        xFountainLogPassBadMsg := TRUE;
    END_IF;
    iFountainLogPinEntry := 0;
END_IF;

tonFountainLogClearedMsg(IN := xFountainLogClearedMsg, PT := T#3S);
IF tonFountainLogClearedMsg.Q THEN xFountainLogClearedMsg := FALSE; END_IF;

tonFountainLogPassBadMsg(IN := xFountainLogPassBadMsg, PT := T#3S);
IF tonFountainLogPassBadMsg.Q THEN xFountainLogPassBadMsg := FALSE; END_IF;

IF xFountainLogClear THEN
    FOR iClearIdx := 1 TO 60 DO
        aFountainLog[iClearIdx] := "";
    END_FOR;
    iFountainLogCount    := 0;
    xFountainLogClear     := FALSE;
    xAskClearFountainLog  := FALSE;
END_IF;

IF xPumpLogPinSubmit THEN
    xPumpLogPinSubmit := FALSE;
    IF iPumpLogPinEntry = iAdminPassCorrect THEN
        GVL.xLogClear       := TRUE;
        GVL.xAskClearLog    := FALSE;
        xPumpLogClearedMsg  := TRUE;
    ELSE
        xPumpLogPassBadMsg := TRUE;
    END_IF;
    iPumpLogPinEntry := 0;
END_IF;

tonPumpLogClearedMsg(IN := xPumpLogClearedMsg, PT := T#3S);
IF tonPumpLogClearedMsg.Q THEN xPumpLogClearedMsg := FALSE; END_IF;

tonPumpLogPassBadMsg(IN := xPumpLogPassBadMsg, PT := T#3S);
IF tonPumpLogPassBadMsg.Q THEN xPumpLogPassBadMsg := FALSE; END_IF;

IF NOT xFountainLogInitialized THEN
    iLogPrevPumpSelect          := iPumpSelect;
    iLogPrevLightSelect         := iLightSelect;
    xLogPrevVseSist             := xVseSist;
    iLogPrevLightScheduleMode   := iLightScheduleMode;
    iLogPrevPumpScheduleMode    := iPumpScheduleMode;
    iLogPrevLightOnHourWeekday   := iLightOnHourWeekday;
    iLogPrevLightOnMinuteWeekday := iLightOnMinuteWeekday;
    iLogPrevLightOnHourWeekend   := iLightOnHourWeekend;
    iLogPrevLightOnMinuteWeekend := iLightOnMinuteWeekend;
    iLogPrevPumpOnHourWeekday    := iPumpOnHourWeekday;
    iLogPrevPumpOnMinuteWeekday  := iPumpOnMinuteWeekday;
    iLogPrevPumpOnHourWeekend    := iPumpOnHourWeekend;
    iLogPrevPumpOnMinuteWeekend  := iPumpOnMinuteWeekend;
    iLogPrevOffHourWeekday       := iOffHourWeekday;
    iLogPrevOffMinuteWeekday     := iOffMinuteWeekday;
    iLogPrevOffHourWeekend       := iOffHourWeekend;
    iLogPrevOffMinuteWeekend     := iOffMinuteWeekend;
    iLogPrevSunsetCorrectSigned  := iSunsetCorrectSigned;
    iLogPrevChoseTimeZone        := iChoseTimeZone;
    rLogPrevSunLatitude          := rSunLatitude;
    rLogPrevSunLongitude         := rSunLongitude;
    iLogPrevFilterMinRunMin      := iFilterMinRunMin;
    xLogPrevAlarmReset           := xAlarmReset;
    xFountainLogInitialized      := TRUE;
END_IF;

IF iPumpSelect <> iLogPrevPumpSelect THEN
    F_FountainLogWrite(WCONCAT("Режим насосов: ", WCONCAT(F_SelectModeText(iLogPrevPumpSelect), WCONCAT(" → ", F_SelectModeText(iPumpSelect)))));
    iLogPrevPumpSelect := iPumpSelect;
END_IF;

IF iLightSelect <> iLogPrevLightSelect THEN
    F_FountainLogWrite(WCONCAT("Режим света: ", WCONCAT(F_SelectModeText(iLogPrevLightSelect), WCONCAT(" → ", F_SelectModeText(iLightSelect)))));
    iLogPrevLightSelect := iLightSelect;
END_IF;

IF xVseSist <> xLogPrevVseSist THEN
    F_FountainLogWrite(WCONCAT("Общее разрешение: ", WCONCAT(SEL(xLogPrevVseSist, "Запрещено", "Разрешено"), WCONCAT(" → ", SEL(xVseSist, "Запрещено", "Разрешено")))));
    xLogPrevVseSist := xVseSist;
END_IF;

IF iLightScheduleMode <> iLogPrevLightScheduleMode THEN
    F_FountainLogWrite(WCONCAT("Расписание света: ", WCONCAT(F_LightScheduleModeText(iLogPrevLightScheduleMode), WCONCAT(" → ", F_LightScheduleModeText(iLightScheduleMode)))));
    iLogPrevLightScheduleMode := iLightScheduleMode;
END_IF;

IF iPumpScheduleMode <> iLogPrevPumpScheduleMode THEN
    F_FountainLogWrite(WCONCAT("Расписание насосов: ", WCONCAT(F_PumpScheduleModeText(iLogPrevPumpScheduleMode), WCONCAT(" → ", F_PumpScheduleModeText(iPumpScheduleMode)))));
    iLogPrevPumpScheduleMode := iPumpScheduleMode;
END_IF;

IF iLightOnHourWeekday <> iLogPrevLightOnHourWeekday THEN
    F_FountainLogWrite(WCONCAT("Свет вкл будние дни, час: ", WCONCAT(INT_TO_WSTRING(iLogPrevLightOnHourWeekday), WCONCAT(" → ", INT_TO_WSTRING(iLightOnHourWeekday)))));
    iLogPrevLightOnHourWeekday := iLightOnHourWeekday;
END_IF;
IF iLightOnMinuteWeekday <> iLogPrevLightOnMinuteWeekday THEN
    F_FountainLogWrite(WCONCAT("Свет вкл будние дни, мин: ", WCONCAT(INT_TO_WSTRING(iLogPrevLightOnMinuteWeekday), WCONCAT(" → ", INT_TO_WSTRING(iLightOnMinuteWeekday)))));
    iLogPrevLightOnMinuteWeekday := iLightOnMinuteWeekday;
END_IF;
IF iLightOnHourWeekend <> iLogPrevLightOnHourWeekend THEN
    F_FountainLogWrite(WCONCAT("Свет вкл выходные дни, час: ", WCONCAT(INT_TO_WSTRING(iLogPrevLightOnHourWeekend), WCONCAT(" → ", INT_TO_WSTRING(iLightOnHourWeekend)))));
    iLogPrevLightOnHourWeekend := iLightOnHourWeekend;
END_IF;
IF iLightOnMinuteWeekend <> iLogPrevLightOnMinuteWeekend THEN
    F_FountainLogWrite(WCONCAT("Свет вкл выходные дни, мин: ", WCONCAT(INT_TO_WSTRING(iLogPrevLightOnMinuteWeekend), WCONCAT(" → ", INT_TO_WSTRING(iLightOnMinuteWeekend)))));
    iLogPrevLightOnMinuteWeekend := iLightOnMinuteWeekend;
END_IF;

IF iPumpOnHourWeekday <> iLogPrevPumpOnHourWeekday THEN
    F_FountainLogWrite(WCONCAT("Насосы вкл будние дни, час: ", WCONCAT(INT_TO_WSTRING(iLogPrevPumpOnHourWeekday), WCONCAT(" → ", INT_TO_WSTRING(iPumpOnHourWeekday)))));
    iLogPrevPumpOnHourWeekday := iPumpOnHourWeekday;
END_IF;
IF iPumpOnMinuteWeekday <> iLogPrevPumpOnMinuteWeekday THEN
    F_FountainLogWrite(WCONCAT("Насосы вкл будние дни, мин: ", WCONCAT(INT_TO_WSTRING(iLogPrevPumpOnMinuteWeekday), WCONCAT(" → ", INT_TO_WSTRING(iPumpOnMinuteWeekday)))));
    iLogPrevPumpOnMinuteWeekday := iPumpOnMinuteWeekday;
END_IF;
IF iPumpOnHourWeekend <> iLogPrevPumpOnHourWeekend THEN
    F_FountainLogWrite(WCONCAT("Насосы вкл выходные дни, час: ", WCONCAT(INT_TO_WSTRING(iLogPrevPumpOnHourWeekend), WCONCAT(" → ", INT_TO_WSTRING(iPumpOnHourWeekend)))));
    iLogPrevPumpOnHourWeekend := iPumpOnHourWeekend;
END_IF;
IF iPumpOnMinuteWeekend <> iLogPrevPumpOnMinuteWeekend THEN
    F_FountainLogWrite(WCONCAT("Насосы вкл выходные дни, мин: ", WCONCAT(INT_TO_WSTRING(iLogPrevPumpOnMinuteWeekend), WCONCAT(" → ", INT_TO_WSTRING(iPumpOnMinuteWeekend)))));
    iLogPrevPumpOnMinuteWeekend := iPumpOnMinuteWeekend;
END_IF;

IF iOffHourWeekday <> iLogPrevOffHourWeekday THEN
    F_FountainLogWrite(WCONCAT("Выкл фонтана будние дни, час: ", WCONCAT(INT_TO_WSTRING(iLogPrevOffHourWeekday), WCONCAT(" → ", INT_TO_WSTRING(iOffHourWeekday)))));
    iLogPrevOffHourWeekday := iOffHourWeekday;
END_IF;
IF iOffMinuteWeekday <> iLogPrevOffMinuteWeekday THEN
    F_FountainLogWrite(WCONCAT("Выкл фонтана будние дни, мин: ", WCONCAT(INT_TO_WSTRING(iLogPrevOffMinuteWeekday), WCONCAT(" → ", INT_TO_WSTRING(iOffMinuteWeekday)))));
    iLogPrevOffMinuteWeekday := iOffMinuteWeekday;
END_IF;
IF iOffHourWeekend <> iLogPrevOffHourWeekend THEN
    F_FountainLogWrite(WCONCAT("Выкл фонтана выходные дни, час: ", WCONCAT(INT_TO_WSTRING(iLogPrevOffHourWeekend), WCONCAT(" → ", INT_TO_WSTRING(iOffHourWeekend)))));
    iLogPrevOffHourWeekend := iOffHourWeekend;
END_IF;
IF iOffMinuteWeekend <> iLogPrevOffMinuteWeekend THEN
    F_FountainLogWrite(WCONCAT("Выкл фонтана выходные дни, мин: ", WCONCAT(INT_TO_WSTRING(iLogPrevOffMinuteWeekend), WCONCAT(" → ", INT_TO_WSTRING(iOffMinuteWeekend)))));
    iLogPrevOffMinuteWeekend := iOffMinuteWeekend;
END_IF;

IF iSunsetCorrectSigned <> iLogPrevSunsetCorrectSigned THEN
    F_FountainLogWrite(WCONCAT("Коррекция заката: ", WCONCAT(INT_TO_WSTRING(iLogPrevSunsetCorrectSigned), WCONCAT(" → ", WCONCAT(INT_TO_WSTRING(iSunsetCorrectSigned), ", мин")))));
    iLogPrevSunsetCorrectSigned := iSunsetCorrectSigned;
END_IF;

IF iChoseTimeZone <> iLogPrevChoseTimeZone THEN
    F_FountainLogWrite(WCONCAT("Часовой пояс: ", WCONCAT(INT_TO_WSTRING(iLogPrevChoseTimeZone), WCONCAT(" → ", INT_TO_WSTRING(iChoseTimeZone)))));
    iLogPrevChoseTimeZone := iChoseTimeZone;
END_IF;

IF rSunLatitude <> rLogPrevSunLatitude THEN
    F_FountainLogWrite(WCONCAT("Широта: ", WCONCAT(REAL_TO_WSTRING(rLogPrevSunLatitude), WCONCAT(" → ", REAL_TO_WSTRING(rSunLatitude)))));
    rLogPrevSunLatitude := rSunLatitude;
END_IF;

IF rSunLongitude <> rLogPrevSunLongitude THEN
    F_FountainLogWrite(WCONCAT("Долгота: ", WCONCAT(REAL_TO_WSTRING(rLogPrevSunLongitude), WCONCAT(" → ", REAL_TO_WSTRING(rSunLongitude)))));
    rLogPrevSunLongitude := rSunLongitude;
END_IF;

IF iFilterMinRunMin <> iLogPrevFilterMinRunMin THEN
    F_FountainLogWrite(WCONCAT("Порог подтв.режима НФ: ", WCONCAT(INT_TO_WSTRING(iLogPrevFilterMinRunMin), WCONCAT(" → ", WCONCAT(INT_TO_WSTRING(iFilterMinRunMin), ", мин")))));
    iLogPrevFilterMinRunMin := iFilterMinRunMin;
END_IF;

IF xAlarmReset AND NOT xLogPrevAlarmReset THEN
    F_FountainLogWrite("Сброс всех аварий");
END_IF;
xLogPrevAlarmReset := xAlarmReset;

(* ============================================================ *)
(* 14. ОБЩИЕ СТРОКОВЫЕ СТАТУСЫ                                   *)
(* ============================================================ *)
IF xVseSist THEN sVseSistStatus := "Разрешен"; ELSE sVseSistStatus := "Запрещен"; END_IF;
xPermissionToWork := xVseSist AND NOT xDryRunAlarm;

(* ============================================================ *)
(* 15. ЗАПИСЬ ВЫХОДОВ DO — НОВАЯ КАРТА (ТОЛЬКО 4 ВЫХОДА)          *)
(* ============================================================ *)
xDO[1]  := xDryRunOk;      // DO1 — дубляж сухого хода (=DI4)
xDO[2]  := xPumpsCmd;      // DO2 — пуск насосов фонтана
xDO[3]  := xLightCmd;      // DO3 — пуск подсветки
xDO[4]  := xDamperCmdRaw;  // DO4 — дубляж клапана добора (=DI5)
xDO[5]  := FALSE;
xDO[6]  := FALSE;
xDO[7]  := FALSE;
xDO[8]  := FALSE;
xDO[9]  := FALSE;
xDO[10] := FALSE;
xDO[11] := FALSE;
xDO[12] := FALSE;
xDO[13] := FALSE;
xDO[14] := FALSE;
xDO[15] := FALSE;
xDO[16] := FALSE;

(* ---- PRG_IO.st ---- *)
(* ============================================================ *)
(* PRG_IO — распаковка входов МВ110, сборка выходов МУ110       *)
(* === 60ЛО: НОВАЯ КАРТА ("60 Лет Октября") ===                 *)
(*                                                              *)
(* КАРТА DI (МВ110-16Д):                                       *)
(*   DI1  ПЧ1 (насос-шоу, информационный, ни на что не влияет) *)
(*   DI2  ПЧ2 (насос-шоу, информационный)                      *)
(*   DI3  ПЧ3 (насос-шоу, информационный, НОВЫЙ)                *)
(*   DI4  Сухой ход от Мусидоры (1=норма)                       *)
(*   DI5  Пуск добора от Мусидоры (автоматика, мы не решаем)    *)
(*   DI6  Подтверждение положения клапана добора                *)
(*   DI7  Контактор фильтрации (НФ физически работает)          *)
(*   DI8  Подтверждение реле сухого хода                        *)
(*   DI9  Подтверждение работы насосов фонтана                  *)
(*   DI10 Подтверждение работы подсветки                        *)
(*   DI11 Ручка режима фильтрации = АВТО                        *)
(*   DI12 Ручка режима фильтрации = РУЧНОЙ                      *)
(*                                                              *)
(* КАРТА DO (МУ110-16Р):                                       *)
(*   DO1  дубляж сухого хода (=DI4)                             *)
(*   DO2  пуск насосов фонтана                                  *)
(*   DO3  пуск подсветки                                        *)
(*   DO4  дубляж клапана добора (=DI5)                          *)
(*   DO5..DO16 — свободны                                       *)
(* Семантическая распаковка DI и сборка DO — в PRG_Fountain     *)
(* (блоки 2 и 15). Здесь только упаковка/распаковка сырых        *)
(* массивов xDI[]/xDO[], логика тела программы НЕ МЕНЯЛАСЬ.      *)
(* ============================================================ *)
PROGRAM PRG_IO
VAR
    i : INT;
    tonMU110SafeInit   : TON;
    xMU110SafeInitDone : BOOL := FALSE;
    tonMV110Hold       : TON;          // удержание входов при сбое связи МВ110
    tDI_Hold           : TIME := T#10S; // время удержания входов
END_VAR
(* Безопасное состояние МУ110: через 3 сек после старта         *)
(* однократно взводим триггер записи (все выходы=0 при потере   *)
(* связи мастер↔МУ110).                                         *)
tonMU110SafeInit(IN := NOT xMU110SafeInitDone, PT := T#3S);
IF tonMU110SafeInit.Q AND NOT xMU110SafeInitDone THEN
    xMU110_WriteSafe   := TRUE;
    xMU110SafeInitDone := TRUE;
ELSE
    xMU110_WriteSafe := FALSE;
END_IF;

(* Входы МВ110 → xDI[1..16]. Удержание последнего значения при   *)
(* кратком сбое связи (tDI_Hold). Логика не меняется.          *)
tonMV110Hold(IN := xMV110_Error, PT := tDI_Hold);

IF xMV110_Error AND tonMV110Hold.Q THEN
    FOR i := 1 TO cDI_Count DO
        xDI[i] := FALSE;
    END_FOR;
ELSIF NOT xMV110_Error THEN
    FOR i := 1 TO cDI_Count DO
        xDI[i] := (wMV110_Inputs AND SHL(WORD#1, INT_TO_BYTE(i - 1))) <> WORD#0;
    END_FOR;
END_IF;

(* Распаковка семантических DI делается в PRG_Fountain блок 2.  *)
(* Здесь только заполняем массив xDI[].                          *)

(* Выходы xDO[1..16] → маска МУ110. При потере связи — 0.       *)
IF xMU110_Error THEN
    wMU110_Outputs := 0;
ELSE
    wMU110_Outputs := 0;
    FOR i := 1 TO cDO_Count DO
        IF xDO[i] THEN
            wMU110_Outputs := wMU110_Outputs OR SHL(WORD#1, INT_TO_BYTE(i - 1));
        END_IF;
    END_FOR;
END_IF;

(* ---- PRG_IO_Write.st ---- *)
(* ============================================================ *)
(* PRG_IO_Write — СБОРКА маски выходов МУ110 из xDO[]           *)
(* === 60ЛО:НОВЫЙ POU === Выделен из PRG_IO, чтобы устранить     *)
(* задержку на 1 скан. Вызывается в PLC_PRG ПОСЛЕ PRG_Fountain,  *)
(* поэтому xDO[] здесь — уже посчитанные значения ЭТОГО цикла.   *)
(*                                                              *)
(* Логика полностью перенесена из старого PRG_IO без изменений:  *)
(* при потере связи с МУ110 маска = 0 (все выходы выключены).    *)
(* ============================================================ *)
PROGRAM PRG_IO_Write
VAR
    i : INT;
END_VAR

(* Выходы xDO[1..16] → маска МУ110. При потере связи — 0. *)
IF xMU110_Error THEN
    wMU110_Outputs := 0;
ELSE
    wMU110_Outputs := 0;
    FOR i := 1 TO cDO_Count DO
        IF xDO[i] THEN
            wMU110_Outputs := wMU110_Outputs OR SHL(WORD#1, INT_TO_BYTE(i - 1));
        END_IF;
    END_FOR;
END_IF;

(* ---- PRG_Pumps.st ---- *)
PROGRAM PRG_Pumps
(* ============================================================ *)
(* === 60ЛО: почти без изменений относительно ДДЮТ ===           *)
(* ПЧ на COM2 (адреса 41/42/43) качают насосы-шоу — вся механика  *)
(* отладки RS-485, чтения/записи параметров, журнала и разовой    *)
(* инициализации работает одинаково независимо от их назначения.  *)
(* === 60ЛО:ИСПРАВЛЕНО (баг) === Блок 4а был жёстко прописан      *)
(* только на 2 насоса (EMD_PUMP_1/EMD_PUMP_2) — при cPumpCount=3   *)
(* третий насос вообще не проверялся бы на обрыв связи. Добавлен   *)
(* EMD_PUMP_3. ВАЖНО: устройство EMD_PUMP_3 нужно добавить в       *)
(* дереве Modbus проекта (по аналогии с EMD_PUMP_1/2, адрес 43)    *)
(* — без него этот файл не скомпилируется.                         *)
(* ============================================================ *)
VAR
    i                       : INT;
    xDebugForPump           : BOOL;
    wActualFaultReg         : WORD;
    iDebugPumpSelected_Prev : INT := 1;
    iPrevDebugMode          : INT := -1;
    tonApplyHold   : ARRAY[1..cPumpCount] OF TON;
    tonFactoryHold : ARRAY[1..cPumpCount] OF TON;
    tApplyHold     : TIME := T#5S;
    tonHoldRead     : ARRAY[1..cPumpCount] OF TON;
    tonHold_AccTime : ARRAY[1..cPumpCount] OF TON;
    tonHold_DecTime : ARRAY[1..cPumpCount] OF TON;
    tonHold_MaxFreq : ARRAY[1..cPumpCount] OF TON;
    tonHold_MinFreq : ARRAY[1..cPumpCount] OF TON;
    tonHold_MotorCur : ARRAY[1..cPumpCount] OF TON;
    tonHold_MotorVolt : ARRAY[1..cPumpCount] OF TON;
    tonHold_OCLevel : ARRAY[1..cPumpCount] OF TON;
    tonHold_OCTime  : ARRAY[1..cPumpCount] OF TON;
    tonHold_OVProt  : ARRAY[1..cPumpCount] OF TON;
    tonHold_Overheat : ARRAY[1..cPumpCount] OF TON;
    tonHold_OCAcc   : ARRAY[1..cPumpCount] OF TON;
    tonHold_F800    : ARRAY[1..cPumpCount] OF TON;
    tonHold_Sources : ARRAY[1..cPumpCount] OF TON;
    tonHold_DispParam : ARRAY[1..cPumpCount] OF TON;
    tonHold_ErrDelay  : ARRAY[1..cPumpCount] OF TON;
    tonInitDelay      : TON;
    xInitDone         : BOOL := FALSE;
    tonStopWait     : ARRAY[1..cPumpCount] OF TON;
    tonStopWaitAll  : ARRAY[1..cPumpCount] OF TON;
    tStopWaitMax    : TIME := T#30S;
    rMaxDecTime     : REAL;
    tWriteHoldDyn   : TIME;
    xNeedStopWrite  : ARRAY[1..cPumpCount] OF BOOL;
    xNoStopWrite    : ARRAY[1..cPumpCount] OF BOOL;
END_VAR
(* ========================================================= *)
(* БЛОК 0а: СИНХРОНИЗАЦИЯ ФЛАГОВ ПРИ СМЕНЕ РЕЖИМА ОТЛАДКИ    *)
(* ========================================================= *)
IF iDebugMode <> iPrevDebugMode THEN
    FOR i := 1 TO cPumpCount DO
        xDebugModePump[i] := FALSE;
    END_FOR;
    xDebugModeAll := FALSE;

    CASE iDebugMode OF
        0: ;
        1: xDebugModePump[iDebugPumpSelected] := TRUE;
        2:
            FOR i := 1 TO cPumpCount DO
                xDebugModePump[i] := TRUE;
            END_FOR;
            xDebugModeAll := TRUE;
    END_CASE;
    iPrevDebugMode := iDebugMode;
END_IF;

(* ========================================================= *)
(* БЛОК 0б: СМЕНА ВЫБРАННОГО НАСОСА                          *)
(* ========================================================= *)
IF (iDebugMode = 1) AND (iDebugPumpSelected <> iDebugPumpSelected_Prev) THEN
    FOR i := 1 TO cPumpCount DO
        xDebugModePump[i] := (i = iDebugPumpSelected);
    END_FOR;
END_IF;
iDebugPumpSelected_Prev := iDebugPumpSelected;

(* ========================================================= *)
(* БЛОК 0в: ОКНО "ПРИМЕНИТЬ ПАРАМЕТРЫ"                       *)
(* ========================================================= *)
IF xDlgConfirmApply THEN
    CASE iDebugMode OF
        0: ;
        1:
            xApplyParamsPump[iDebugPumpSelected] := TRUE;
        2:
            FOR i := 1 TO cPumpCount DO
                rPumpFreqSetHz[i]             := rPumpFreqSetHz[iDebugPumpSelected];
                rPumpAccTime_Set[i]           := rPumpAccTime_Set[iDebugPumpSelected];
                rPumpDecTime_Set[i]           := rPumpDecTime_Set[iDebugPumpSelected];
                rPumpMaxFreq_Set[i]           := rPumpMaxFreq_Set[iDebugPumpSelected];
                rPumpMinFreq_Set[i]           := rPumpMinFreq_Set[iDebugPumpSelected];
                rPumpMotorRatedCurrent_Set[i] := rPumpMotorRatedCurrent_Set[iDebugPumpSelected];
                rPumpMotorRatedVoltage_Set[i] := rPumpMotorRatedVoltage_Set[iDebugPumpSelected];
                rPumpOverCurrentLevel_A_Set[i] := rPumpOverCurrentLevel_A_Set[iDebugPumpSelected];
                rPumpOverCurrentTime_Set[i]   := rPumpOverCurrentTime_Set[iDebugPumpSelected];
                xPumpOverVoltProtect_Set[i]   := xPumpOverVoltProtect_Set[iDebugPumpSelected];
                iPumpOverheatLevel_Set[i]     := iPumpOverheatLevel_Set[iDebugPumpSelected];
                iPumpOverCurAcc_Set[i]        := iPumpOverCurAcc_Set[iDebugPumpSelected];
                xApplyParamsPump[i] := TRUE;
            END_FOR;
    END_CASE;
    xDlgConfirmApply := FALSE;
    xAskApply        := FALSE;
END_IF;

(* ========================================================= *)
(* БЛОК 0г: ОКНО "СБРОС НА ЗАВОДСКИЕ"                        *)
(* ========================================================= *)
IF xDlgConfirmFactory THEN
    CASE iDebugMode OF
        0: ;
        1: xFactoryResetPump[iDebugPumpSelected] := TRUE;
        2: xFactoryResetAll := TRUE;
    END_CASE;
    xDlgConfirmFactory := FALSE;
    xAskFactory        := FALSE;
END_IF;

(* ========================================================= *)
(* БЛОК 0д: ГРУППОВЫЕ ПУСК/СТОП ИЗ visuDebug                 *)
(* ========================================================= *)
IF xDbgRunAll THEN
    FOR i := 1 TO cPumpCount DO
        xPumpRunCmd[i] := TRUE;
    END_FOR;
    xDbgRunAll := FALSE;
END_IF;
IF xDbgStopAll THEN
    FOR i := 1 TO cPumpCount DO
        xPumpRunCmd[i] := FALSE;
    END_FOR;
    xDbgStopAll := FALSE;
END_IF;

(* ========================================================= *)
(* БЛОК 0е: ЧТЕНИЕ ВСЕХ ПАРАМЕТРОВ (кнопка "Считать все")    *)
(* ========================================================= *)
IF xReadAllAsk THEN
    CASE iDebugMode OF
        0:  xReadAllPump[iDebugPumpSelected] := TRUE;
        1: xReadAllPump[iDebugPumpSelected] := TRUE;
        2:
            FOR i := 1 TO cPumpCount DO
                xReadAllPump[i] := TRUE;
            END_FOR;
    END_CASE;
    xReadAllAsk := FALSE;
END_IF;

(* ========================================================= *)
(* БЛОК 0ж: ЗАПИСЬ ВСЕХ ПАРАМЕТРОВ (кнопка "Записать все")    *)
(* ========================================================= *)
IF xWriteAllConfirm THEN
    CASE iDebugMode OF
        0: ;
        1: xWritePending[iDebugPumpSelected] := TRUE;
        2:
            FOR i := 1 TO cPumpCount DO
                xWritePending[i] := TRUE;
            END_FOR;
    END_CASE;
    xWriteAllConfirm := FALSE;
END_IF;

(* ============================================================ *)
(* ЗАПИСЬ ВСЕХ ПАРАМЕТРОВ — через Modbus-стоп (источник RS-485)*)
(* ============================================================ *)
FOR i := 1 TO cPumpCount DO
    IF xWritePending[i] THEN
        wCmdSourceWrite[i]  := WORD#2;
        wFreqSourceWrite[i] := WORD#5;
        xWr_Sources[i]      := TRUE;

        xPumpRunCmd[i] := FALSE;
        tonStopWaitAll[i](IN := TRUE, PT := tStopWaitMax);

        IF xPumpFullyStopped[i] THEN
            tonStopWaitAll[i](IN := FALSE);
            xWr_UnlockF800[i]   := TRUE;
            xWr_AccTime[i]      := TRUE;
            xWr_DecTime[i]      := TRUE;
            xWr_MaxFreq[i]      := TRUE;
            xWr_MinFreq[i]      := TRUE;
            xWr_MotorCurrent[i] := TRUE;
            xWr_MotorVoltage[i] := TRUE;
            xWr_OverCurLevel[i] := TRUE;
            xWr_OverCurTime[i]  := TRUE;
            xWr_OverVoltProt[i] := TRUE;
            xWr_Overheat[i]     := TRUE;
            xWr_OverCurAcc[i]   := TRUE;
            xWritePending[i]    := FALSE;
        ELSIF tonStopWaitAll[i].Q THEN
            xWritePending[i] := FALSE;
            tonStopWaitAll[i](IN := FALSE);
        END_IF;
    END_IF;
END_FOR;

(* ========================================================= *)
(* БЛОК 0з: ЗАПИСЬ ОДНОГО ПАРАМЕТРА (кнопки у строк)         *)
(* ========================================================= *)
rMaxDecTime := 0.0;
FOR i := 1 TO cPumpCount DO
    IF rPumpDecTime_Set[i] > rMaxDecTime THEN
        rMaxDecTime := rPumpDecTime_Set[i];
    END_IF;
END_FOR;
tWriteHoldDyn := REAL_TO_TIME((rMaxDecTime + 5.0) * 1000.0);

FOR i := 1 TO cPumpCount DO
    xNeedStopWrite[i] := xWr_MaxFreq[i] OR xWr_MinFreq[i]
        OR xWr_MotorCurrent[i] OR xWr_MotorVoltage[i] OR xWr_OverCurLevel[i]
        OR xWr_OverCurTime[i] OR xWr_OverVoltProt[i] OR xWr_Overheat[i]
        OR xWr_OverCurAcc[i];

    xNoStopWrite[i] := xWr_AccTime[i] OR xWr_DecTime[i];

    IF xNeedStopWrite[i] OR xNoStopWrite[i] THEN
        xWr_UnlockF800[i] := TRUE;
    END_IF;

    IF xNeedStopWrite[i] THEN
        wCmdSourceWrite[i]  := WORD#2;
        wFreqSourceWrite[i] := WORD#5;
        xWr_Sources[i]      := TRUE;

        IF NOT xPumpFullyStopped[i] THEN
            xPumpRunCmd[i] := FALSE;
            xWaitStopForWrite[i] := TRUE;
			xAskDialogStopPch  := TRUE;
        ELSE
            xWaitStopForWrite[i] := FALSE;
			xAskDialogStopPch  := FALSE;
        END_IF;
    ELSE
        xWaitStopForWrite[i] := FALSE;
    END_IF;
END_FOR;

(* ========================================================= *)
(* БЛОК 1: ГРУППОВОЙ ФЛАГ ОТЛАДКИ                            *)
(* ========================================================= *)
IF xDebugModeAll <> xDebugModeAll_Prev THEN
    FOR i := 1 TO cPumpCount DO
        xDebugModePump[i] := xDebugModeAll;
    END_FOR;
    xDebugModeAll_Prev := xDebugModeAll;
END_IF;

(* ========================================================= *)
(* БЛОК 2: ПЕРЕХВАТ СМЕНЫ РЕЖИМА ОТЛАДКИ — ИСТОЧНИК RS-485   *)
(* ========================================================= *)
FOR i := 1 TO cPumpCount DO
    IF xDebugModePump[i] <> xDebugModePump_Prev[i] THEN
        IF xDebugModePump[i] THEN
            wCmdSourceWrite[i]  := WORD#2;
            wFreqSourceWrite[i] := WORD#5;
        ELSE
            wCmdSourceWrite[i]  := WORD#1;
            wFreqSourceWrite[i] := WORD#3;
        END_IF;
        xWr_Sources[i] := TRUE;
        xDebugModePump_Prev[i] := xDebugModePump[i];
    END_IF;
END_FOR;

(* ========================================================= *)
(* БЛОК 3: ГРУППОВОЙ ТРИГГЕР "ПРИМЕНИТЬ"                     *)
(* ========================================================= *)
IF xApplyParamsAll THEN
    FOR i := 1 TO cPumpCount DO
        xApplyParamsPump[i] := TRUE;
    END_FOR;
    xApplyParamsAll := FALSE;
END_IF;

(* ========================================================= *)
(* БЛОК 4: ГРУППОВОЙ ТРИГГЕР "СБРОС НА ЗАВОДСКИЕ"            *)
(* ========================================================= *)
IF xFactoryResetAll THEN
    FOR i := 1 TO cPumpCount DO
        xFactoryResetPump[i] := TRUE;
    END_FOR;
    xFactoryResetAll := FALSE;
END_IF;

FOR i := 1 TO cPumpCount DO
    IF xFactoryResetPump[i] THEN
        wPumpFactoryResetWrite[i] := WORD#8;
    ELSE
        wPumpFactoryResetWrite[i] := WORD#0;
    END_IF;
END_FOR;

(* ========================================================= *)
(* БЛОК 4а: КОНТРОЛЬ СВЯЗИ — xError + ФИЛЬТР                  *)
(* === 60ЛО:ИСПРАВЛЕНО (баг) === Добавлен EMD_PUMP_3 — раньше   *)
(* здесь были жёстко прописаны только 2 насоса, третий не         *)
(* проверялся бы на обрыв связи вообще. Устройство EMD_PUMP_3     *)
(* нужно добавить в дереве Modbus проекта (адрес 43).              *)
(* ========================================================= *)
xPumpCommRaw[1] := EMD_PUMP_1.xError;
xPumpCommRaw[2] := EMD_PUMP_2.xError;
xPumpCommRaw[3] := EMD_PUMP_3.xError;

tonPumpCommFilter[1](IN := EMD_PUMP_1.xError, PT := T#3S);
xPumpCommError[1] := tonPumpCommFilter[1].Q;

tonPumpCommFilter[2](IN := EMD_PUMP_2.xError, PT := T#3S);
xPumpCommError[2] := tonPumpCommFilter[2].Q;

tonPumpCommFilter[3](IN := EMD_PUMP_3.xError, PT := T#3S);
xPumpCommError[3] := tonPumpCommFilter[3].Q;

(* ========================================================= *)
(* БЛОК 5: ВЫЗОВ FB ДЛЯ ВСЕХ НАСОСОВ                         *)
(* ========================================================= *)
FOR i := 1 TO cPumpCount DO
    xDebugForPump   := xDebugModePump[i] OR xDebugModeAll;
    wActualFaultReg := wPumpFaultReg[i];

    Pump[i](
        eType                  := ePumpType[i],
        xDebugMode             := xDebugForPump,
        xCommError             := xPumpCommError[i],
        xCommUnstable          := xPumpCommRaw[i],

        xRunCmd                := xPumpRunCmd[i],
        rFreqSetHz             := rPumpFreqSetHz[i],

        wStatus                := wPumpStatus[i],
        wFaultReg              := wActualFaultReg,
        wFreqSetRead           := wPumpFreqSetRead[i],
        wFreqActual            := wPumpFreqActual[i],
        wCurrentActual         := wPumpCurrentActual[i],
        wSpeedActual           := wPumpSpeedActual[i],
        wDcVoltage             := wPumpDcVoltage[i],
        wTemperature           := wPumpTemperature[i],
        wVoltageActual         := wPumpVoltageActual[i],
        wRuntimeHoursRaw       := wPumpRuntimeHoursRaw[i],
        wAccTimeRawRead        := wPumpAccTimeRaw[i],
        wDecTimeRawRead        := wPumpDecTimeRaw[i],
        wMaxFreqRead           := wPumpMaxFreqRead[i],
        wMinFreqRead           := wPumpMinFreqRead[i],
        wMotorRatedCurrentRead := wPumpMotorRatedCurrentRead[i],
        wMotorRatedVoltageRead := wPumpMotorRatedVoltageRead[i],
        wOverCurrentLevelRead  := wPumpOverCurrentLevelRead[i],
        wOverheatLevelRead     := wPumpOverheatLevelRead[i],
        wOverCurAccRead        := wPumpOverCurAccRead[i],
        wOverCurrentTimeRead   := wPumpOverCurrentTimeRead[i],
        wOverVoltProtectRead   := wPumpOverVoltProtectRead[i],

        rAccTime_Set            := rPumpAccTime_Set[i],
        rDecTime_Set            := rPumpDecTime_Set[i],
        rMaxFreq_Set            := rPumpMaxFreq_Set[i],
        rMinFreq_Set            := rPumpMinFreq_Set[i],
        rMotorRatedCurrent_Set  := rPumpMotorRatedCurrent_Set[i],
        rMotorRatedVoltage_Set  := rPumpMotorRatedVoltage_Set[i],
        rOverCurrentLevel_A_Set := rPumpOverCurrentLevel_A_Set[i],
        rOverCurrentTime_Set    := rPumpOverCurrentTime_Set[i],
        xOverVoltProtect_Set    := xPumpOverVoltProtect_Set[i],
        iOverheatLevel_Set      := iPumpOverheatLevel_Set[i],
        iOverCurAcc_Set         := iPumpOverCurAcc_Set[i],

        wCmd                    => wPumpCmd[i],
        wFreq                   => wPumpFreq[i],
        wAccTimeRawWrite        => wPumpAccTimeWrite[i],
        wDecTimeRawWrite        => wPumpDecTimeWrite[i],
        wMaxFreqWrite           => wPumpMaxFreqWrite[i],
        wMinFreqWrite           => wPumpMinFreqWrite[i],
        wMotorRatedCurrentWrite => wPumpMotorRatedCurrentWrite[i],
        wMotorRatedVoltageWrite => wPumpMotorRatedVoltageWrite[i],
        wOverCurrentLevelWrite  => wPumpOverCurrentLevelWrite[i],
        wOverCurrentTimeWrite   => wPumpOverCurrentTimeWrite[i],
        wOverVoltProtectWrite   => wPumpOverVoltProtectWrite[i],
        wOverheatLevelWrite     => wPumpOverheatLevelWrite[i],
        wOverCurAccWrite        => wPumpOverCurAccWrite[i],

        xRun                    => xPumpWork[i],
        xStop                   => xPumpStop[i],
        xAlarm                  => xPumpAlarm[i],
        sState                  => sPumpState[i],
        sFaultText              => sPumpFaultText[i],
        sTypeText               => sPumpTypeText[i],
        xReverse                => xPumpReverse[i],

        rFreqSetActHz           => rPumpFreqSetActHz[i],
        rFreqActHz              => rPumpFreqActHz[i],
        rCurrentActA            => rPumpCurrentActA[i],
        rSpeedActRpm            => rPumpSpeedActRpm[i],
        rDcVoltageV             => rPumpDcVoltageV[i],
        iTemperatureC           => iPumpTemperatureC[i],
        rVoltageActV            => rPumpVoltageActV[i],
        rRuntimeHours           => rPumpRuntimeHours[i],
        rAccTime_Disp            => rPumpAccTime_Disp[i],
        rDecTime_Disp            => rPumpDecTime_Disp[i],
        rMaxFreq_Disp            => rPumpMaxFreq_Disp[i],
        rMinFreq_Disp            => rPumpMinFreq_Disp[i],
        rMotorRatedCurrent_Disp  => rPumpMotorRatedCurrent_Disp[i],
        rMotorRatedVoltage_Disp  => rPumpMotorRatedVoltage_Disp[i],
        rOverCurrentLevel_A_Disp => rPumpOverCurrentLevel_A_Disp[i],
        iOverCurrentLevel_pct_Disp => iPumpOverCurrentLevel_pct_Disp[i],
        iOverheatLevel_Disp      => iPumpOverheatLevel_Disp[i],
        iOverCurAcc_Disp         => iPumpOverCurAcc_Disp[i],
        rOverCurrentTime_Disp    => rPumpOverCurrentTime_Disp[i],
        xOverVoltProtect_Disp    => xPumpOverVoltProtect_Disp[i]
    );

    IF xPumpCommError[i] OR xPumpCommRaw[i] THEN
        dwPumpLampColor[i] := OVD.COLORS.OwenKeyGrey;
    ELSIF xPumpAlarm[i] THEN
        dwPumpLampColor[i] := OVD.COLORS.Red;
    ELSIF xPumpWork[i] THEN
        dwPumpLampColor[i] := OVD.COLORS.Green;
    ELSE
        dwPumpLampColor[i] := OVD.COLORS.OwenKeyGrey;
    END_IF;
    rPumpFreqPresetHz[i] := WORD_TO_REAL(wPumpFreqPresetRead[i]) / 100.0;
END_FOR;

(* ========================================================= *)
(* БЛОК 5_СТОП: ПРИЗНАК "ПЧ ПОЛНОСТЬЮ ОСТАНОВЛЕН"           *)
(* ========================================================= *)
FOR i := 1 TO cPumpCount DO
    IF xPumpCommError[i] THEN
        xPumpFullyStopped[i] := FALSE;
    ELSE
        xPumpFullyStopped[i] :=
            ((wPumpStatus[i] AND 16#0001) = WORD#0)
            AND (wPumpFreqActual[i] = WORD#0);
    END_IF;
END_FOR;

(* ========================================================= *)
(* БЛОК 5а: РАСШИФРОВКА ИСТОРИИ АВАРИЙ                       *)
(* ========================================================= *)
FOR i := 1 TO cPumpCount DO
    IF xPumpCommError[i] THEN
        sPumpFaultText[i]     := "Задержка связи";
        sPumpFaultLastText[i] := "Задержка связи";
        sPumpFault2Text[i]    := "Задержка связи";
        sPumpFault3Text[i]    := "Задержка связи";
        sPumpFault4Text[i]    := "Задержка связи";
    ELSE
        IF (wPumpFaultLast[i] AND 16#7FFF) = WORD#0 THEN
            sPumpFaultLastText[i] := "Нет аварии";
        ELSE
            sPumpFaultLastText[i] := F_FaultCodeToText(ePumpType[i], wPumpFaultLast[i]);
        END_IF;
        IF (wPumpFault2[i] AND 16#7FFF) = WORD#0 THEN
            sPumpFault2Text[i] := "Нет аварии";
        ELSE
            sPumpFault2Text[i] := F_FaultCodeToText(ePumpType[i], wPumpFault2[i]);
        END_IF;
        IF (wPumpFault3[i] AND 16#7FFF) = WORD#0 THEN
            sPumpFault3Text[i] := "Нет аварии";
        ELSE
            sPumpFault3Text[i] := F_FaultCodeToText(ePumpType[i], wPumpFault3[i]);
        END_IF;
        IF (wPumpFault4[i] AND 16#7FFF) = WORD#0 THEN
            sPumpFault4Text[i] := "Нет аварии";
        ELSE
            sPumpFault4Text[i] := F_FaultCodeToText(ePumpType[i], wPumpFault4[i]);
        END_IF;
    END_IF;
END_FOR;

(* ========================================================= *)
(* БЛОК 5б: ТЕКСТ СТАТУСА ЗАЩИТЫ ПЕРЕНАПРЯЖЕНИЯ              *)
(* ========================================================= *)
FOR i := 1 TO cPumpCount DO
    IF xPumpOverVoltProtect_Disp[i] THEN
        sPumpOverVoltProtect[i] := "Включена";
    ELSE
        sPumpOverVoltProtect[i] := "Выключена";
    END_IF;
END_FOR;

(* ========================================================= *)
(* БЛОК 6: РАЗБЛОКИРОВКА РАСШИРЕННЫХ НАСТРОЕК (F800)         *)
(* ========================================================= *)
FOR i := 1 TO cPumpCount DO
    IF xWr_UnlockF800[i] THEN
        wPumpExtSettingsUnlockWrite[i] := WORD#1;
    ELSE
        wPumpExtSettingsUnlockWrite[i] := WORD#0;
    END_IF;
END_FOR;

(* ========================================================= *)
(* БЛОК 7: УДЕРЖАНИЕ ВСЕХ ТРИГГЕРОВ (таймаут tApplyHold)      *)
(* ========================================================= *)
FOR i := 1 TO cPumpCount DO
    tonHoldRead[i](IN := xReadAllPump[i], PT := tApplyHold);
    IF tonHoldRead[i].Q THEN xReadAllPump[i] := FALSE; tonHoldRead[i](IN := FALSE); END_IF;

    tonHold_AccTime[i](IN := xWr_AccTime[i], PT := tApplyHold);
    IF tonHold_AccTime[i].Q THEN xWr_AccTime[i] := FALSE; tonHold_AccTime[i](IN := FALSE); END_IF;

    tonHold_DecTime[i](IN := xWr_DecTime[i], PT := tApplyHold);
    IF tonHold_DecTime[i].Q THEN xWr_DecTime[i] := FALSE; tonHold_DecTime[i](IN := FALSE); END_IF;

    tonHold_MaxFreq[i](IN := xWr_MaxFreq[i], PT := tWriteHoldDyn);
    IF tonHold_MaxFreq[i].Q THEN xWr_MaxFreq[i] := FALSE; tonHold_MaxFreq[i](IN := FALSE); END_IF;

    tonHold_MinFreq[i](IN := xWr_MinFreq[i], PT := tWriteHoldDyn);
    IF tonHold_MinFreq[i].Q THEN xWr_MinFreq[i] := FALSE; tonHold_MinFreq[i](IN := FALSE); END_IF;

    tonHold_MotorCur[i](IN := xWr_MotorCurrent[i], PT := tWriteHoldDyn);
    IF tonHold_MotorCur[i].Q THEN xWr_MotorCurrent[i] := FALSE; tonHold_MotorCur[i](IN := FALSE); END_IF;

    tonHold_MotorVolt[i](IN := xWr_MotorVoltage[i], PT := tWriteHoldDyn);
    IF tonHold_MotorVolt[i].Q THEN xWr_MotorVoltage[i] := FALSE; tonHold_MotorVolt[i](IN := FALSE); END_IF;

    tonHold_OCLevel[i](IN := xWr_OverCurLevel[i], PT := tWriteHoldDyn);
    IF tonHold_OCLevel[i].Q THEN xWr_OverCurLevel[i] := FALSE; tonHold_OCLevel[i](IN := FALSE); END_IF;

    tonHold_OCTime[i](IN := xWr_OverCurTime[i], PT := tWriteHoldDyn);
    IF tonHold_OCTime[i].Q THEN xWr_OverCurTime[i] := FALSE; tonHold_OCTime[i](IN := FALSE); END_IF;

    tonHold_OVProt[i](IN := xWr_OverVoltProt[i], PT := tWriteHoldDyn);
    IF tonHold_OVProt[i].Q THEN xWr_OverVoltProt[i] := FALSE; tonHold_OVProt[i](IN := FALSE); END_IF;

    tonHold_Overheat[i](IN := xWr_Overheat[i], PT := tWriteHoldDyn);
    IF tonHold_Overheat[i].Q THEN xWr_Overheat[i] := FALSE; tonHold_Overheat[i](IN := FALSE); END_IF;

    tonHold_OCAcc[i](IN := xWr_OverCurAcc[i], PT := tWriteHoldDyn);
    IF tonHold_OCAcc[i].Q THEN xWr_OverCurAcc[i] := FALSE; tonHold_OCAcc[i](IN := FALSE); END_IF;

    tonHold_F800[i](IN := xWr_UnlockF800[i], PT := tWriteHoldDyn);
    IF tonHold_F800[i].Q THEN xWr_UnlockF800[i] := FALSE; tonHold_F800[i](IN := FALSE); END_IF;

    tonHold_Sources[i](IN := xWr_Sources[i], PT := tApplyHold);
    IF tonHold_Sources[i].Q THEN xWr_Sources[i] := FALSE; tonHold_Sources[i](IN := FALSE); END_IF;

    tonHold_DispParam[i](IN := xWr_DispParam[i], PT := tApplyHold);
    IF tonHold_DispParam[i].Q THEN xWr_DispParam[i] := FALSE; tonHold_DispParam[i](IN := FALSE); END_IF;

    tonHold_ErrDelay[i](IN := xWr_ErrDelayInit[i], PT := tApplyHold);
    IF tonHold_ErrDelay[i].Q THEN xWr_ErrDelayInit[i] := FALSE; tonHold_ErrDelay[i](IN := FALSE); END_IF;

    tonFactoryHold[i](IN := xFactoryResetPump[i], PT := tApplyHold);
    IF tonFactoryHold[i].Q THEN xFactoryResetPump[i] := FALSE; tonFactoryHold[i](IN := FALSE); END_IF;

    tonApplyHold[i](IN := xApplyParamsPump[i], PT := tApplyHold);
    IF tonApplyHold[i].Q THEN xApplyParamsPump[i] := FALSE; tonApplyHold[i](IN := FALSE); END_IF;
END_FOR;

(* ========================================================= *)
(* БЛОК 8: ЖУРНАЛ ИЗМЕНЕНИЙ ПАРАМЕТРОВ ПЧ                    *)
(* ========================================================= *)
IF xLogClear THEN
    FOR i := 1 TO 30 DO
        aPumpLog[i] := "";
    END_FOR;
    iPumpLogCount  := 0;
    xLogClear      := FALSE;
    xAskClearLog   := FALSE;   (* PLC сам закрывает диалог. *)
    (* GVL.xLogClear пишется ТОЛЬКО из PRG_Fountain.st (блок проверки  *)
    (* пароля через СВОЙ экран) — см. переменные xPumpLogPinEntry/     *)
    (* xPumpLogPinSubmit там же. Сама очистка и закрытие диалога        *)
    (* остаются здесь.                                                  *)
END_IF;

FOR i := 1 TO cPumpCount DO

    IF xPumpCommError[i] THEN
        xLog_Initialized[i] := FALSE;
    END_IF;

    IF rtrigReadAll_Prev[i] AND NOT xReadAllPump[i] AND NOT xPumpCommError[i] THEN
        rLog_AccTime_Prev[i]   := rPumpAccTime_Disp[i];
        rLog_DecTime_Prev[i]   := rPumpDecTime_Disp[i];
        rLog_MaxFreq_Prev[i]   := rPumpMaxFreq_Disp[i];
        rLog_MinFreq_Prev[i]   := rPumpMinFreq_Disp[i];
        rLog_MotorCur_Prev[i]  := rPumpMotorRatedCurrent_Disp[i];
        rLog_MotorVolt_Prev[i] := rPumpMotorRatedVoltage_Disp[i];
        rLog_OCLevel_Prev[i]   := rPumpOverCurrentLevel_A_Disp[i];
        rLog_OCTime_Prev[i]    := rPumpOverCurrentTime_Disp[i];
        xLog_OVProt_Prev[i]    := xPumpOverVoltProtect_Disp[i];
        iLog_Overheat_Prev[i]  := iPumpOverheatLevel_Disp[i];
        iLog_OCAcc_Prev[i]     := iPumpOverCurAcc_Disp[i];
        xLog_Initialized[i]    := TRUE;
    END_IF;
    rtrigReadAll_Prev[i] := xReadAllPump[i];

    IF NOT xPumpCommError[i] AND xLog_Initialized[i] THEN

        IF rPumpAccTime_Disp[i] <> rLog_AccTime_Prev[i] THEN
            F_PumpLogWrite(WCONCAT(F_FormatLogTimestamp(),
                WCONCAT(" | ПЧ", WCONCAT(INT_TO_WSTRING(i),
                WCONCAT(" | Разгон: ", WCONCAT(REAL_TO_WSTRING(rLog_AccTime_Prev[i]),
                WCONCAT("→", WCONCAT(REAL_TO_WSTRING(rPumpAccTime_Disp[i]), "с$N"))))))));
            rLog_AccTime_Prev[i] := rPumpAccTime_Disp[i];
        END_IF;

        IF rPumpDecTime_Disp[i] <> rLog_DecTime_Prev[i] THEN
            F_PumpLogWrite(WCONCAT(F_FormatLogTimestamp(),
                WCONCAT(" | ПЧ", WCONCAT(INT_TO_WSTRING(i),
                WCONCAT(" | Торможение: ", WCONCAT(REAL_TO_WSTRING(rLog_DecTime_Prev[i]),
                WCONCAT("→", WCONCAT(REAL_TO_WSTRING(rPumpDecTime_Disp[i]), "с$N"))))))));
            rLog_DecTime_Prev[i] := rPumpDecTime_Disp[i];
        END_IF;

        IF rPumpMaxFreq_Disp[i] <> rLog_MaxFreq_Prev[i] THEN
            F_PumpLogWrite(WCONCAT(F_FormatLogTimestamp(),
                WCONCAT(" | ПЧ", WCONCAT(INT_TO_WSTRING(i),
                WCONCAT(" | Макс.част: ", WCONCAT(REAL_TO_WSTRING(rLog_MaxFreq_Prev[i]),
                WCONCAT("→", WCONCAT(REAL_TO_WSTRING(rPumpMaxFreq_Disp[i]), "Гц$N"))))))));
            rLog_MaxFreq_Prev[i] := rPumpMaxFreq_Disp[i];
        END_IF;

        IF rPumpMinFreq_Disp[i] <> rLog_MinFreq_Prev[i] THEN
            F_PumpLogWrite(WCONCAT(F_FormatLogTimestamp(),
                WCONCAT(" | ПЧ", WCONCAT(INT_TO_WSTRING(i),
                WCONCAT(" | Мин.част: ", WCONCAT(REAL_TO_WSTRING(rLog_MinFreq_Prev[i]),
                WCONCAT("→", WCONCAT(REAL_TO_WSTRING(rPumpMinFreq_Disp[i]), "Гц$N"))))))));
            rLog_MinFreq_Prev[i] := rPumpMinFreq_Disp[i];
        END_IF;

        IF rPumpMotorRatedCurrent_Disp[i] <> rLog_MotorCur_Prev[i] THEN
            F_PumpLogWrite(WCONCAT(F_FormatLogTimestamp(),
                WCONCAT(" | ПЧ", WCONCAT(INT_TO_WSTRING(i),
                WCONCAT(" | Ном.ток: ", WCONCAT(REAL_TO_WSTRING(rLog_MotorCur_Prev[i]),
                WCONCAT("→", WCONCAT(REAL_TO_WSTRING(rPumpMotorRatedCurrent_Disp[i]), "А$N"))))))));
            rLog_MotorCur_Prev[i] := rPumpMotorRatedCurrent_Disp[i];
        END_IF;

        IF rPumpMotorRatedVoltage_Disp[i] <> rLog_MotorVolt_Prev[i] THEN
            F_PumpLogWrite(WCONCAT(F_FormatLogTimestamp(),
                WCONCAT(" | ПЧ", WCONCAT(INT_TO_WSTRING(i),
                WCONCAT(" | Ном.напр: ", WCONCAT(REAL_TO_WSTRING(rLog_MotorVolt_Prev[i]),
                WCONCAT("→", WCONCAT(REAL_TO_WSTRING(rPumpMotorRatedVoltage_Disp[i]), "В$N"))))))));
            rLog_MotorVolt_Prev[i] := rPumpMotorRatedVoltage_Disp[i];
        END_IF;

        IF rPumpOverCurrentLevel_A_Disp[i] <> rLog_OCLevel_Prev[i] THEN
            F_PumpLogWrite(WCONCAT(F_FormatLogTimestamp(),
                WCONCAT(" | ПЧ", WCONCAT(INT_TO_WSTRING(i),
                WCONCAT(" | Ур.тока: ", WCONCAT(REAL_TO_WSTRING(rLog_OCLevel_Prev[i]),
                WCONCAT("→", WCONCAT(REAL_TO_WSTRING(rPumpOverCurrentLevel_A_Disp[i]), "А$N"))))))));
            rLog_OCLevel_Prev[i] := rPumpOverCurrentLevel_A_Disp[i];
        END_IF;

        IF rPumpOverCurrentTime_Disp[i] <> rLog_OCTime_Prev[i] THEN
            F_PumpLogWrite(WCONCAT(F_FormatLogTimestamp(),
                WCONCAT(" | ПЧ", WCONCAT(INT_TO_WSTRING(i),
                WCONCAT(" | Вр.тока: ", WCONCAT(REAL_TO_WSTRING(rLog_OCTime_Prev[i]),
                WCONCAT("→", WCONCAT(REAL_TO_WSTRING(rPumpOverCurrentTime_Disp[i]), "с$N"))))))));
            rLog_OCTime_Prev[i] := rPumpOverCurrentTime_Disp[i];
        END_IF;

        IF xPumpOverVoltProtect_Disp[i] <> xLog_OVProt_Prev[i] THEN
            F_PumpLogWrite(WCONCAT(F_FormatLogTimestamp(),
                WCONCAT(" | ПЧ", WCONCAT(INT_TO_WSTRING(i),
                WCONCAT(" | Зщт.перенапр: ", WCONCAT(SEL(xLog_OVProt_Prev[i], "Выкл", "Вкл"),
                WCONCAT("→", WCONCAT(SEL(xPumpOverVoltProtect_Disp[i], "Выкл", "Вкл"), "$N"))))))));
            xLog_OVProt_Prev[i] := xPumpOverVoltProtect_Disp[i];
        END_IF;

        IF iPumpOverheatLevel_Disp[i] <> iLog_Overheat_Prev[i] THEN
            F_PumpLogWrite(WCONCAT(F_FormatLogTimestamp(),
                WCONCAT(" | ПЧ", WCONCAT(INT_TO_WSTRING(i),
                WCONCAT(" | Перегрев: ", WCONCAT(INT_TO_WSTRING(iLog_Overheat_Prev[i]),
                WCONCAT("→", WCONCAT(INT_TO_WSTRING(iPumpOverheatLevel_Disp[i]), "°C$N"))))))));
            iLog_Overheat_Prev[i] := iPumpOverheatLevel_Disp[i];
        END_IF;

        IF iPumpOverCurAcc_Disp[i] <> iLog_OCAcc_Prev[i] THEN
            F_PumpLogWrite(WCONCAT(F_FormatLogTimestamp(),
                WCONCAT(" | ПЧ", WCONCAT(INT_TO_WSTRING(i),
                WCONCAT(" | Огр.тока.разг: ", WCONCAT(INT_TO_WSTRING(iLog_OCAcc_Prev[i]),
                WCONCAT("→", WCONCAT(INT_TO_WSTRING(iPumpOverCurAcc_Disp[i]), "%$N"))))))));
            iLog_OCAcc_Prev[i] := iPumpOverCurAcc_Disp[i];
        END_IF;

    END_IF;
END_FOR;

(* ========================================================= *)
(* БЛОК 9: РАЗОВАЯ ИНИЦИАЛИЗАЦИЯ ПАРАМЕТРОВ ПЧ ПРИ СТАРТЕ    *)
(* ========================================================= *)
tonInitDelay(IN := TRUE, PT := T#5S);

IF tonInitDelay.Q AND NOT xInitDone THEN
    FOR i := 1 TO cPumpCount DO
        IF NOT xErrDelayWritten[i] AND NOT xPumpCommError[i] THEN
            wPumpRS_ErrDelayWrite[i] := WORD#5;
            xWr_ErrDelayInit[i]      := TRUE;
            xErrDelayWritten[i]      := TRUE;
        END_IF;

        IF NOT xDispParamWritten[i] AND NOT xPumpCommError[i] THEN
            wPumpDispParamWrite[i] := WORD#1;
            xWr_DispParam[i]       := TRUE;
            xDispParamWritten[i]   := TRUE;
        END_IF;
    END_FOR;
    xInitDone := TRUE;
END_IF;

(* ---- PRG_TimeCorrect.st ---- *)
(* ============================================================ *)
(* PRG_TimeCorrect — КОРРЕКЦИЯ УХОДА СИСТЕМНЫХ ЧАСОВ (RTC)      *)
(* ============================================================ *)
(* RTC контроллера уходит вперёд. Один раз в НОВЫЙ календарный    *)
(* день (как только сменился iCurrentDay) отводим RTC назад на    *)
(* iTimeDriftCorrSec секунд. Час/минута НЕ важны — сработает при   *)
(* первом же скане нового дня, даже если питание пропадало.       *)
(*                                                              *)
(* iLastCorrDay — RETAIN: переживает перезагрузку, поэтому после   *)
(* рестарта в тот же день коррекция повторно НЕ сработает          *)
(* (ровно 1 раз в сутки, а не на каждый ребут).                  *)
(*                                                              *)
(* Ставить время из приложения ПЛК МОЖНО — не защищённая          *)
(* операция. Вызывается в PLC_PRG ПОСЛЕ PRG_Fountain.             *)
(*                                                              *)
(* Сигнатура (подтверждена по библиотеке SysTimeRtc проекта):     *)
(*   SysTimeRtcSet(ulTimestamp : DWORD) : RTS_IEC_RESULT          *)
(*   (Seconds since 1.1.1970 00:00 UTC).                          *)
(* ============================================================ *)
PROGRAM PRG_TimeCorrect
VAR RETAIN
    iLastCorrDay : INT := -1;   // день месяца последней коррекции (RETAIN — 1 раз в сутки, переживает ребут)
END_VAR
VAR
    dwUtcRaw   : DWORD;
    rtcRes     : DWORD;
    xDoCorrect : BOOL;
END_VAR

(* --- Когда корректировать --- *)
xDoCorrect := FALSE;

(* Авто: раз в новый день, НАЧИНАЯ с часа iTimeDriftCorrHour.        *)
(* Минута НЕ проверяется (окно — весь день от этого часа), поэтому    *)
(* пропуск из-за пропадания питания не страшен: сработает на первом   *)
(* же скане после включения, если день новый и час уже наступил.      *)
(* ⚠️ Час нужен, чтобы вычитание секунд НЕ пересекало полночь: без    *)
(* него (чистый «новый день») коррекция в 00:00 откатывает время в    *)
(* 23:59 прошлого дня → день снова «новый» → бесконечный откат, часы   *)
(* залипают на полуночи. iTimeDriftCorrHour>=1 (0 не ставить!).        *)
IF xTimeDriftCorrEnable
   AND (iCurrentDay <> iLastCorrDay)
   AND (iCurrentHour >= iTimeDriftCorrHour) THEN
    xDoCorrect := TRUE;
END_IF;

(* Ручной триггер с экрана — срабатывает один раз *)
IF xTimeDriftCorrNow THEN
    xDoCorrect := TRUE;
END_IF;

(* --- Собственно коррекция --- *)
IF xDoCorrect THEN
    (* Читаем СЫРОЕ UTC (без смещения пояса!), вычитаем N секунд, пишем обратно *)
    dwUtcRaw := SysTimeRtcGet(pResult := rtcRes);
    dwUtcRaw := dwUtcRaw - INT_TO_DWORD(iTimeDriftCorrSec);
    rtcRes   := SysTimeRtcSet(dwUtcRaw);

    iLastCorrDay        := iCurrentDay;
    iTimeDriftCorrCount := iTimeDriftCorrCount + 1;
    sTimeDriftLast      := sCurrentDateStr;   // дата последней коррекции для экрана
    xTimeDriftCorrNow   := FALSE;             // гасим ручной триггер
END_IF;

(* iTimeDriftCorrHour — час-якорь (по умолч. 3), с которого в новый    *)
(* день разрешена коррекция. НЕ ставить 0 (см. предупреждение выше).    *)
(* iTimeDriftCorrSec — на сколько секунд отводить назад (по умолч. 15;  *)
(* поставь 20, если измеренный уход ~20с/сутки).                        *)
